Yaskawa INFORM job: DEMO_ROOF_SIDE_0625_3PAINT_5.JBI

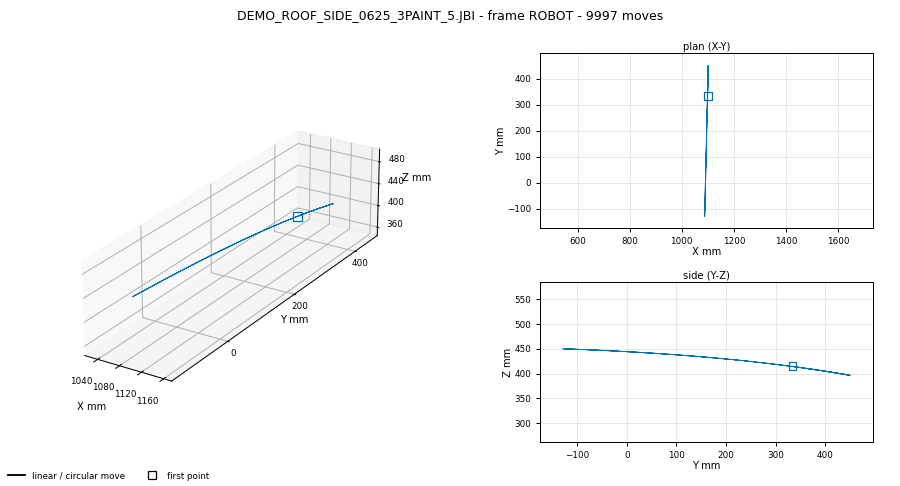
[picture p0: tool path of DEMO_ROOF_SIDE_0625_3PAINT_5.JBI in frame ROBOT, 9997 of 9997 moves have a stored position in this frame; points joined in program order, loops and branches not executed]
/JOB
//NAME DEMO_ROOF_SIDE_0625_3PAINT5
//POS
///NPOS 9997,0,0,0,0,0
///TOOL 0
///USER 0
///POSTYPE ROBOT
///RECTAN
///RCONF 1,0,0,0,0,0,0,0,0,0,0,0,0,0,0,0,0,0,0,0,0,0,0,0
C00000=1099.831,334.377,414.802,179.080,18.325,152.124
C00001=1099.836,334.624,414.769,179.083,18.328,152.124
C00002=1099.842,334.872,414.736,179.086,18.331,152.124
C00003=1099.847,335.120,414.703,179.089,18.334,152.124
C00004=1099.853,335.368,414.670,179.092,18.337,152.124
C00005=1099.859,335.615,414.637,179.095,18.340,152.124
C00006=1099.865,335.863,414.604,179.099,18.343,152.124
C00007=1099.870,336.112,414.571,179.102,18.346,152.125
C00008=1099.876,336.359,414.539,179.105,18.349,152.125
C00009=1099.881,336.607,414.505,179.109,18.352,152.125
C00010=1099.887,336.855,414.472,179.112,18.355,152.125
C00011=1099.893,337.102,414.439,179.115,18.358,152.125
C00012=1099.899,337.350,414.406,179.118,18.361,152.125
C00013=1099.904,337.598,414.372,179.121,18.364,152.125
C00014=1099.910,337.845,414.338,179.124,18.367,152.125
C00015=1099.916,338.093,414.306,179.127,18.370,152.125
C00016=1099.922,338.341,414.272,179.131,18.373,152.126
C00017=1099.928,338.589,414.239,179.134,18.376,152.126
C00018=1099.933,338.837,414.206,179.137,18.379,152.126
C00019=1099.939,339.084,414.172,179.140,18.382,152.126
C00020=1099.945,339.332,414.140,179.143,18.385,152.126
C00021=1099.951,339.580,414.106,179.146,18.388,152.126
C00022=1099.956,339.827,414.072,179.150,18.392,152.127
C00023=1099.961,340.074,414.039,179.153,18.395,152.127
C00024=1099.967,340.322,414.006,179.156,18.397,152.127
C00025=1099.972,340.570,413.973,179.159,18.401,152.127
C00026=1099.978,340.818,413.939,179.162,18.404,152.127
C00027=1099.984,341.065,413.905,179.165,18.407,152.127
C00028=1099.989,341.313,413.872,179.168,18.411,152.128
C00029=1099.996,341.561,413.839,179.171,18.413,152.128
C00030=1100.001,341.809,413.806,179.175,18.417,152.128
C00031=1100.007,342.056,413.772,179.178,18.420,152.128
C00032=1100.013,342.304,413.738,179.181,18.423,152.128
C00033=1100.018,342.552,413.705,179.184,18.427,152.128
C00034=1100.027,342.925,413.654,179.189,18.431,152.129
C00035=1100.036,343.298,413.603,179.194,18.436,152.129
C00036=1100.044,343.671,413.552,179.199,18.441,152.129
C00037=1100.053,344.044,413.502,179.203,18.446,152.129
C00038=1100.059,344.291,413.469,179.207,18.449,152.130
C00039=1100.065,344.539,413.435,179.209,18.452,152.130
C00040=1100.070,344.787,413.401,179.212,18.455,152.130
C00041=1100.076,345.034,413.367,179.216,18.459,152.130
C00042=1100.082,345.283,413.333,179.219,18.462,152.130
C00043=1100.087,345.530,413.299,179.222,18.466,152.131
C00044=1100.093,345.778,413.266,179.225,18.469,152.131
C00045=1100.099,346.025,413.231,179.228,18.472,152.131
C00046=1100.104,346.273,413.198,179.231,18.475,152.131
C00047=1100.110,346.520,413.164,179.234,18.479,152.132
C00048=1100.116,346.768,413.130,179.238,18.482,152.132
C00049=1100.121,347.016,413.097,179.240,18.486,152.132
C00050=1100.127,347.263,413.062,179.244,18.489,152.132
C00051=1100.132,347.511,413.029,179.247,18.492,152.132
C00052=1100.138,347.758,412.995,179.249,18.495,152.133
C00053=1100.144,348.006,412.960,179.253,18.499,152.133
C00054=1100.150,348.254,412.926,179.256,18.502,152.133
C00055=1100.156,348.502,412.893,179.259,18.506,152.133
C00056=1100.161,348.749,412.858,179.262,18.509,152.134
C00057=1100.167,348.997,412.824,179.265,18.513,152.134
C00058=1100.172,349.244,412.791,179.268,18.516,152.134
C00059=1100.178,349.492,412.757,179.272,18.520,152.134
C00060=1100.184,349.740,412.722,179.274,18.523,152.135
C00061=1100.190,349.987,412.688,179.278,18.527,152.135
C00062=1100.196,350.235,412.654,179.281,18.530,152.135
C00063=1100.201,350.482,412.619,179.284,18.534,152.135
C00064=1100.206,350.730,412.586,179.287,18.537,152.136
C00065=1100.212,350.977,412.552,179.290,18.541,152.136
C00066=1100.219,351.225,412.517,179.293,18.544,152.136
C00067=1100.224,351.473,412.483,179.296,18.548,152.136
C00068=1100.230,351.720,412.448,179.299,18.551,152.137
C00069=1100.236,351.967,412.414,179.302,18.555,152.137
C00070=1100.241,352.215,412.380,179.305,18.558,152.137
C00071=1100.247,352.463,412.345,179.309,18.562,152.138
C00072=1100.253,352.710,412.311,179.311,18.565,152.138
C00073=1100.258,352.958,412.277,179.315,18.569,152.138
C00074=1100.264,353.205,412.243,179.318,18.572,152.139
C00075=1100.270,353.454,412.208,179.321,18.577,152.139
C00076=1100.276,353.701,412.174,179.323,18.580,152.139
C00077=1100.281,353.948,412.139,179.327,18.584,152.139
C00078=1100.287,354.196,412.105,179.329,18.587,152.140
C00079=1100.293,354.444,412.070,179.333,18.591,152.140
C00080=1100.298,354.691,412.036,179.336,18.594,152.140
C00081=1100.304,354.939,412.002,179.339,18.598,152.141
C00082=1100.309,355.186,411.967,179.342,18.602,152.141
C00083=1100.316,355.434,411.932,179.345,18.606,152.141
C00084=1100.321,355.681,411.897,179.348,18.609,152.142
C00085=1100.327,355.928,411.863,179.351,18.613,152.142
C00086=1100.335,356.304,411.810,179.356,18.619,152.143
C00087=1100.344,356.679,411.758,179.360,18.625,152.143
C00088=1100.353,357.055,411.706,179.365,18.630,152.144
C00089=1100.361,357.430,411.653,179.369,18.636,152.144
C00090=1100.367,357.678,411.618,179.372,18.639,152.144
C00091=1100.373,357.925,411.583,179.375,18.644,152.145
C00092=1100.378,358.172,411.548,179.378,18.647,152.145
C00093=1100.384,358.420,411.514,179.381,18.651,152.146
C00094=1100.390,358.667,411.479,179.385,18.655,152.146
C00095=1100.396,358.914,411.445,179.387,18.659,152.146
C00096=1100.402,359.162,411.409,179.391,18.663,152.147
C00097=1100.407,359.410,411.374,179.393,18.666,152.147
C00098=1100.413,359.658,411.340,179.396,18.670,152.148
C00099=1100.419,359.905,411.304,179.399,18.675,152.148
C00100=1100.425,360.152,411.270,179.402,18.678,152.148
C00101=1100.431,360.400,411.235,179.405,18.682,152.149
C00102=1100.436,360.647,411.200,179.409,18.686,152.149
C00103=1100.441,360.894,411.165,179.411,18.690,152.149
C00104=1100.448,361.142,411.130,179.414,18.694,152.150
C00105=1100.453,361.389,411.095,179.417,18.698,152.150
C00106=1100.459,361.637,411.060,179.420,18.702,152.151
C00107=1100.464,361.884,411.024,179.423,18.706,152.151
C00108=1100.470,362.131,410.990,179.426,18.710,152.152
C00109=1100.476,362.379,410.955,179.429,18.714,152.152
C00110=1100.482,362.626,410.919,179.432,18.718,152.152
C00111=1100.488,362.874,410.884,179.435,18.722,152.153
C00112=1100.493,363.121,410.850,179.438,18.726,152.153
C00113=1100.499,363.369,410.814,179.441,18.730,152.154
C00114=1100.505,363.616,410.778,179.444,18.734,152.154
C00115=1100.510,363.863,410.744,179.447,18.738,152.154
C00116=1100.516,364.111,410.708,179.450,18.743,152.155
C00117=1100.521,364.358,410.673,179.452,18.746,152.155
C00118=1100.528,364.606,410.638,179.456,18.751,152.156
C00119=1100.533,364.853,410.603,179.459,18.755,152.156
C00120=1100.539,365.101,410.567,179.461,18.758,152.157
C00121=1100.545,365.348,410.532,179.464,18.763,152.157
C00122=1100.551,365.595,410.496,179.468,18.767,152.158
C00123=1100.556,365.842,410.461,179.470,18.771,152.158
C00124=1100.562,366.091,410.426,179.473,18.775,152.159
C00125=1100.567,366.338,410.390,179.476,18.780,152.159
C00126=1100.573,366.585,410.355,179.479,18.784,152.160
C00127=1100.579,366.832,410.319,179.482,18.788,152.160
C00128=1100.585,367.080,410.284,179.485,18.792,152.161
C00129=1100.590,367.327,410.248,179.488,18.797,152.161
C00130=1100.596,367.575,410.212,179.490,18.801,152.162
C00131=1100.602,367.822,410.177,179.494,18.805,152.162
C00132=1100.608,368.069,410.141,179.497,18.809,152.163
C00133=1100.613,368.316,410.106,179.500,18.814,152.163
C00134=1100.619,368.564,410.070,179.502,18.818,152.164
C00135=1100.625,368.811,410.035,179.505,18.822,152.164
C00136=1100.631,369.059,409.999,179.508,18.827,152.165
C00137=1100.636,369.306,409.964,179.511,18.832,152.165
C00138=1100.645,369.696,409.908,179.516,18.838,152.166
C00139=1100.654,370.086,409.851,179.520,18.845,152.167
C00140=1100.664,370.476,409.794,179.524,18.852,152.168
C00141=1100.672,370.867,409.738,179.529,18.859,152.169
C00142=1100.678,371.114,409.702,179.532,18.863,152.169
C00143=1100.684,371.362,409.666,179.535,18.867,152.170
C00144=1100.689,371.609,409.631,179.538,18.872,152.170
C00145=1100.695,371.856,409.595,179.541,18.877,152.171
C00146=1100.701,372.103,409.559,179.544,18.881,152.171
C00147=1100.707,372.350,409.524,179.546,18.885,152.172
C00148=1100.712,372.598,409.487,179.549,18.890,152.173
C00149=1100.718,372.845,409.451,179.552,18.895,152.173
C00150=1100.724,373.092,409.415,179.555,18.899,152.174
C00151=1100.730,373.340,409.380,179.558,18.904,152.174
C00152=1100.736,373.586,409.344,179.560,18.908,152.175
C00153=1100.741,373.834,409.307,179.563,18.913,152.176
C00154=1100.747,374.082,409.271,179.566,18.917,152.176
C00155=1100.753,374.329,409.236,179.569,18.922,152.177
C00156=1100.759,374.576,409.200,179.572,18.927,152.177
C00157=1100.764,374.824,409.163,179.575,18.932,152.178
C00158=1100.770,375.071,409.127,179.577,18.936,152.179
C00159=1100.776,375.318,409.091,179.580,18.941,152.179
C00160=1100.781,375.566,409.055,179.583,18.945,152.180
C00161=1100.787,375.812,409.019,179.586,18.950,152.181
C00162=1100.792,376.060,408.982,179.589,18.955,152.181
C00163=1100.799,376.307,408.946,179.592,18.960,152.182
C00164=1100.804,376.554,408.910,179.595,18.965,152.182
C00165=1100.810,376.801,408.873,179.597,18.970,152.183
C00166=1100.816,377.049,408.838,179.600,18.974,152.184
C00167=1100.821,377.296,408.801,179.602,18.979,152.184
C00168=1100.827,377.543,408.765,179.605,18.984,152.185
C00169=1100.832,377.791,408.728,179.608,18.988,152.186
C00170=1100.838,378.037,408.692,179.611,18.993,152.186
C00171=1100.845,378.284,408.656,179.614,18.998,152.187
C00172=1100.850,378.532,408.619,179.617,19.003,152.188
C00173=1100.856,378.779,408.583,179.620,19.008,152.188
C00174=1100.861,379.026,408.546,179.622,19.013,152.189
C00175=1100.867,379.273,408.510,179.625,19.018,152.190
C00176=1100.873,379.521,408.473,179.627,19.022,152.191
C00177=1100.879,379.768,408.437,179.630,19.027,152.191
C00178=1100.884,380.015,408.400,179.633,19.032,152.192
C00179=1100.890,380.262,408.364,179.636,19.037,152.193
C00180=1100.896,380.510,408.328,179.638,19.042,152.193
C00181=1100.902,380.757,408.291,179.641,19.047,152.194
C00182=1100.908,381.004,408.254,179.644,19.052,152.195
C00183=1100.913,381.250,408.218,179.647,19.057,152.196
C00184=1100.919,381.498,408.181,179.649,19.062,152.196
C00185=1100.925,381.745,408.144,179.652,19.068,152.197
C00186=1100.931,381.992,408.107,179.655,19.073,152.198
C00187=1100.937,382.239,408.070,179.658,19.078,152.199
C00188=1100.943,382.487,408.034,179.661,19.083,152.199
C00189=1100.948,382.733,407.997,179.663,19.088,152.200
C00190=1100.958,383.151,407.936,179.668,19.096,152.201
C00191=1100.967,383.568,407.873,179.673,19.105,152.203
C00192=1100.978,383.985,407.811,179.677,19.114,152.204
C00193=1100.987,384.403,407.749,179.682,19.123,152.205
C00194=1100.992,384.650,407.712,179.684,19.128,152.206
C00195=1100.998,384.897,407.675,179.687,19.133,152.207
C00196=1101.004,385.144,407.637,179.689,19.139,152.208
C00197=1101.010,385.391,407.601,179.692,19.144,152.209
C00198=1101.016,385.638,407.564,179.695,19.149,152.209
C00199=1101.021,385.885,407.527,179.697,19.155,152.210
C00200=1101.027,386.133,407.490,179.700,19.160,152.211
C00201=1101.032,386.380,407.453,179.703,19.165,152.212
C00202=1101.038,386.626,407.416,179.705,19.170,152.213
C00203=1101.044,386.873,407.379,179.708,19.176,152.214
C00204=1101.050,387.121,407.342,179.710,19.181,152.214
C00205=1101.055,387.367,407.304,179.713,19.187,152.215
C00206=1101.061,387.615,407.267,179.716,19.192,152.216
C00207=1101.067,387.862,407.230,179.719,19.198,152.217
C00208=1101.073,388.109,407.193,179.721,19.203,152.218
C00209=1101.079,388.356,407.156,179.724,19.209,152.219
C00210=1101.084,388.603,407.119,179.727,19.214,152.220
C00211=1101.090,388.850,407.081,179.729,19.220,152.220
C00212=1101.096,389.097,407.044,179.732,19.225,152.221
C00213=1101.102,389.345,407.007,179.734,19.230,152.222
C00214=1101.108,389.592,406.969,179.737,19.236,152.223
C00215=1101.113,389.839,406.932,179.739,19.242,152.224
C00216=1101.119,390.086,406.895,179.743,19.248,152.225
C00217=1101.125,390.333,406.857,179.745,19.253,152.226
C00218=1101.131,390.579,406.820,179.748,19.258,152.227
C00219=1101.137,390.827,406.783,179.750,19.264,152.228
C00220=1101.143,391.074,406.746,179.753,19.270,152.229
C00221=1101.149,391.320,406.708,179.755,19.276,152.230
C00222=1101.154,391.568,406.671,179.758,19.281,152.230
C00223=1101.160,391.814,406.633,179.761,19.287,152.231
C00224=1101.166,392.062,406.596,179.763,19.293,152.232
C00225=1101.172,392.308,406.558,179.766,19.299,152.233
C00226=1101.178,392.555,406.520,179.768,19.304,152.234
C00227=1101.183,392.803,406.483,179.770,19.310,152.235
C00228=1101.189,393.049,406.446,179.773,19.316,152.236
C00229=1101.194,393.296,406.407,179.776,19.322,152.237
C00230=1101.200,393.544,406.370,179.779,19.327,152.238
C00231=1101.206,393.790,406.332,179.781,19.333,152.239
C00232=1101.212,394.038,406.294,179.783,19.339,152.240
C00233=1101.218,394.285,406.257,179.786,19.345,152.241
C00234=1101.224,394.532,406.220,179.789,19.351,152.242
C00235=1101.229,394.779,406.181,179.791,19.357,152.243
C00236=1101.235,395.026,406.143,179.793,19.363,152.244
C00237=1101.241,395.273,406.106,179.796,19.369,152.245
C00238=1101.246,395.520,406.069,179.799,19.375,152.246
C00239=1101.253,395.767,406.031,179.801,19.381,152.247
C00240=1101.258,396.014,405.992,179.803,19.387,152.248
C00241=1101.264,396.261,405.954,179.806,19.393,152.249
C00242=1101.269,396.476,405.922,179.808,19.398,152.250
C00243=1101.274,396.690,405.889,179.810,19.403,152.251
C00244=1101.279,396.906,405.856,179.812,19.409,152.252
C00245=1101.284,397.121,405.823,179.815,19.415,152.253
C00246=1101.289,397.335,405.789,179.817,19.419,152.254
C00247=1101.294,397.550,405.756,179.819,19.425,152.255
C00248=1101.299,397.765,405.723,179.821,19.430,152.256
C00249=1101.304,397.980,405.690,179.823,19.436,152.257
C00250=1101.309,398.227,405.652,179.825,19.442,152.258
C00251=1101.315,398.473,405.614,179.828,19.448,152.259
C00252=1101.322,398.721,405.576,179.830,19.455,152.260
C00253=1101.327,398.968,405.538,179.833,19.460,152.261
C00254=1101.333,399.215,405.500,179.836,19.467,152.262
C00255=1101.339,399.461,405.462,179.838,19.473,152.264
C00256=1101.344,399.709,405.424,179.840,19.480,152.265
C00257=1101.351,399.955,405.385,179.843,19.486,152.266
C00258=1101.356,400.202,405.347,179.845,19.492,152.267
C00259=1101.362,400.449,405.309,179.847,19.498,152.268
C00260=1101.367,400.697,405.270,179.850,19.506,152.269
C00261=1101.373,400.944,405.232,179.852,19.512,152.271
C00262=1101.378,401.191,405.194,179.854,19.518,152.272
C00263=1101.385,401.437,405.155,179.857,19.525,152.273
C00264=1101.390,401.685,405.117,179.859,19.531,152.274
C00265=1101.396,401.931,405.079,179.862,19.538,152.275
C00266=1101.402,402.179,405.040,179.864,19.544,152.276
C00267=1101.408,402.425,405.002,179.866,19.551,152.278
C00268=1101.414,402.672,404.964,179.869,19.557,152.279
C00269=1101.419,402.920,404.925,179.871,19.564,152.280
C00270=1101.426,403.166,404.886,179.874,19.571,152.281
C00271=1101.431,403.413,404.848,179.876,19.577,152.283
C00272=1101.437,403.660,404.809,179.879,19.584,152.284
C00273=1101.443,403.907,404.771,179.881,19.591,152.285
C00274=1101.448,404.154,404.733,179.884,19.598,152.286
C00275=1101.455,404.401,404.694,179.886,19.604,152.287
C00276=1101.460,404.648,404.655,179.888,19.611,152.289
C00277=1101.466,404.895,404.616,179.891,19.618,152.290
C00278=1101.472,405.142,404.578,179.893,19.625,152.291
C00279=1101.477,405.388,404.539,179.895,19.631,152.292
C00280=1101.483,405.636,404.500,179.898,19.638,152.294
C00281=1101.489,405.882,404.462,179.900,19.645,152.295
C00282=1101.495,406.130,404.423,179.903,19.652,152.296
C00283=1101.500,406.376,404.384,179.905,19.659,152.298
C00284=1101.506,406.623,404.345,179.907,19.666,152.299
C00285=1101.512,406.870,404.307,179.909,19.673,152.300
C00286=1101.518,407.117,404.268,179.912,19.680,152.302
C00287=1101.524,407.364,404.229,179.914,19.687,152.303
C00288=1101.529,407.611,404.190,179.916,19.694,152.304
C00289=1101.535,407.858,404.151,179.919,19.702,152.306
C00290=1101.541,408.104,404.112,179.921,19.708,152.307
C00291=1101.547,408.352,404.074,179.923,19.716,152.309
C00292=1101.553,408.598,404.034,179.925,19.722,152.310
C00293=1101.558,408.845,403.995,179.928,19.730,152.311
C00294=1101.564,409.092,403.956,179.930,19.738,152.313
C00295=1101.569,409.339,403.918,179.932,19.744,152.314
C00296=1101.575,409.586,403.878,179.935,19.752,152.315
C00297=1101.581,409.832,403.839,179.937,19.759,152.317
C00298=1101.587,410.048,403.805,179.939,19.765,152.318
C00299=1101.591,410.263,403.771,179.941,19.772,152.319
C00300=1101.596,410.478,403.737,179.942,19.778,152.321
C00301=1101.601,410.693,403.703,179.945,19.784,152.322
C00302=1101.606,410.906,403.668,179.947,19.791,152.323
C00303=1101.612,411.122,403.634,179.949,19.797,152.324
C00304=1101.616,411.336,403.600,179.950,19.804,152.326
C00305=1101.622,411.552,403.566,179.953,19.810,152.327
C00306=1101.627,411.798,403.527,179.955,19.818,152.328
C00307=1101.633,412.045,403.488,179.957,19.826,152.330
C00308=1101.639,412.292,403.449,179.959,19.833,152.331
C00309=1101.645,412.539,403.409,179.962,19.840,152.333
C00310=1101.651,412.786,403.370,179.964,19.848,152.334
C00311=1101.656,413.032,403.331,179.967,19.856,152.336
C00312=1101.662,413.280,403.291,179.969,19.864,152.337
C00313=1101.667,413.526,403.252,179.971,19.871,152.339
C00314=1101.673,413.773,403.212,179.973,19.879,152.340
C00315=1101.680,414.020,403.172,179.975,19.886,152.342
C00316=1101.685,414.266,403.133,179.978,19.894,152.343
C00317=1101.691,414.513,403.094,179.980,19.902,152.345
C00318=1101.697,414.761,403.054,179.982,19.909,152.346
C00319=1101.703,415.006,403.014,179.984,19.917,152.348
C00320=1101.709,415.253,402.975,179.986,19.925,152.350
C00321=1101.715,415.501,402.936,179.989,19.933,152.351
C00322=1101.721,415.747,402.896,179.991,19.941,152.353
C00323=1101.726,415.994,402.856,179.993,19.949,152.354
C00324=1101.732,416.241,402.816,179.995,19.956,152.356
C00325=1101.738,416.487,402.777,179.997,19.964,152.358
C00326=1101.744,416.734,402.737,180.000,19.972,152.359
C00327=1101.750,416.981,402.698,-179.998,19.981,152.361
C00328=1101.755,417.227,402.657,-179.996,19.989,152.362
C00329=1101.761,417.474,402.618,-179.994,19.997,152.364
C00330=1101.767,417.721,402.578,-179.991,20.005,152.366
C00331=1101.772,417.968,402.538,-179.989,20.013,152.367
C00332=1101.779,418.215,402.499,-179.987,20.022,152.369
C00333=1101.785,418.461,402.458,-179.985,20.030,152.371
C00334=1101.790,418.708,402.419,-179.983,20.038,152.372
C00335=1101.796,418.955,402.379,-179.981,20.046,152.374
C00336=1101.802,419.201,402.338,-179.978,20.055,152.376
C00337=1101.808,419.448,402.298,-179.976,20.063,152.378
C00338=1101.813,419.694,402.259,-179.974,20.071,152.379
C00339=1101.819,419.942,402.219,-179.972,20.080,152.381
C00340=1101.825,420.188,402.179,-179.970,20.088,152.383
C00341=1101.832,420.435,402.138,-179.968,20.096,152.385
C00342=1101.836,420.682,402.099,-179.966,20.105,152.386
C00343=1101.843,420.928,402.059,-179.964,20.113,152.388
C00344=1101.848,421.175,402.018,-179.962,20.122,152.390
C00345=1101.855,421.421,401.978,-179.959,20.130,152.392
C00346=1101.860,421.669,401.938,-179.958,20.139,152.393
C00347=1101.866,421.915,401.898,-179.955,20.147,152.395
C00348=1101.872,422.161,401.858,-179.954,20.156,152.397
C00349=1101.878,422.408,401.817,-179.952,20.165,152.399
C00350=1101.884,422.654,401.777,-179.949,20.173,152.401
C00351=1101.890,422.902,401.737,-179.947,20.182,152.402
C00352=1101.896,423.148,401.697,-179.946,20.191,152.404
C00353=1101.901,423.395,401.656,-179.943,20.200,152.406
C00354=1101.906,423.616,401.620,-179.941,20.208,152.408
C00355=1101.911,423.838,401.583,-179.939,20.216,152.410
C00356=1101.917,424.059,401.547,-179.938,20.223,152.411
C00357=1101.922,424.281,401.511,-179.936,20.232,152.413
C00358=1101.927,424.503,401.474,-179.934,20.239,152.415
C00359=1101.932,424.724,401.437,-179.932,20.248,152.416
C00360=1101.938,424.946,401.402,-179.931,20.256,152.418
C00361=1101.943,425.167,401.365,-179.928,20.264,152.420
C00362=1101.949,425.414,401.324,-179.927,20.273,152.422
C00363=1101.955,425.661,401.284,-179.925,20.282,152.424
C00364=1101.960,425.907,401.244,-179.922,20.291,152.426
C00365=1101.966,426.154,401.203,-179.920,20.301,152.428
C00366=1101.972,426.401,401.162,-179.919,20.310,152.430
C00367=1101.978,426.647,401.122,-179.917,20.319,152.432
C00368=1101.984,426.893,401.080,-179.914,20.328,152.434
C00369=1101.989,427.140,401.040,-179.912,20.337,152.436
C00370=1101.996,427.387,401.000,-179.911,20.346,152.438
C00371=1102.001,427.633,400.959,-179.909,20.356,152.440
C00372=1102.007,427.880,400.917,-179.907,20.366,152.442
C00373=1102.013,428.126,400.877,-179.905,20.375,152.444
C00374=1102.019,428.373,400.836,-179.903,20.384,152.446
C00375=1102.025,428.619,400.795,-179.901,20.394,152.448
C00376=1102.031,428.866,400.754,-179.899,20.403,152.450
C00377=1102.037,429.113,400.714,-179.897,20.413,152.452
C00378=1102.043,429.359,400.672,-179.896,20.422,152.454
C00379=1102.048,429.605,400.632,-179.893,20.432,152.456
C00380=1102.054,429.851,400.591,-179.892,20.442,152.458
C00381=1102.060,430.098,400.550,-179.890,20.451,152.460
C00382=1102.066,430.344,400.509,-179.888,20.461,152.463
C00383=1102.072,430.591,400.468,-179.886,20.471,152.465
C00384=1102.078,430.837,400.426,-179.884,20.481,152.467
C00385=1102.083,431.084,400.386,-179.882,20.490,152.469
C00386=1102.089,431.330,400.344,-179.881,20.500,152.471
C00387=1102.095,431.577,400.303,-179.878,20.510,152.473
C00388=1102.101,431.823,400.262,-179.877,20.520,152.475
C00389=1102.107,432.069,400.221,-179.875,20.530,152.478
C00390=1102.112,432.316,400.180,-179.873,20.540,152.480
C00391=1102.118,432.562,400.138,-179.871,20.550,152.482
C00392=1102.125,432.809,400.097,-179.869,20.560,152.484
C00393=1102.130,433.056,400.056,-179.868,20.570,152.487
C00394=1102.136,433.302,400.014,-179.866,20.581,152.489
C00395=1102.142,433.549,399.973,-179.864,20.591,152.491
C00396=1102.148,433.795,399.931,-179.862,20.601,152.494
C00397=1102.154,434.041,399.890,-179.861,20.611,152.496
C00398=1102.160,434.288,399.849,-179.859,20.621,152.498
C00399=1102.165,434.534,399.807,-179.857,20.632,152.500
C00400=1102.171,434.781,399.766,-179.855,20.642,152.503
C00401=1102.177,435.027,399.724,-179.853,20.653,152.505
C00402=1102.183,435.273,399.683,-179.852,20.663,152.508
C00403=1102.189,435.519,399.641,-179.850,20.674,152.510
C00404=1102.194,435.766,399.599,-179.848,20.684,152.512
C00405=1102.200,436.012,399.558,-179.846,20.695,152.515
C00406=1102.206,436.258,399.516,-179.845,20.705,152.517
C00407=1102.213,436.505,399.475,-179.843,20.716,152.520
C00408=1102.218,436.751,399.433,-179.842,20.727,152.522
C00409=1102.224,436.998,399.391,-179.840,20.738,152.524
C00410=1102.233,437.381,399.326,-179.838,20.755,152.528
C00411=1102.242,437.764,399.261,-179.835,20.772,152.532
C00412=1102.251,438.148,399.196,-179.832,20.788,152.536
C00413=1102.260,438.531,399.131,-179.830,20.805,152.540
C00414=1102.266,438.778,399.089,-179.828,20.817,152.542
C00415=1102.273,439.023,399.047,-179.826,20.827,152.545
C00416=1102.278,439.270,399.005,-179.825,20.839,152.548
C00417=1102.284,439.517,398.963,-179.823,20.850,152.550
C00418=1102.291,439.762,398.921,-179.822,20.861,152.553
C00419=1102.297,440.008,398.880,-179.821,20.872,152.555
C00420=1102.302,440.255,398.838,-179.819,20.883,152.558
C00421=1102.309,440.501,398.795,-179.817,20.895,152.560
C00422=1102.314,440.748,398.753,-179.815,20.906,152.563
C00423=1102.320,440.993,398.711,-179.814,20.917,152.566
C00424=1102.325,441.240,398.669,-179.813,20.929,152.568
C00425=1102.332,441.487,398.627,-179.811,20.940,152.571
C00426=1102.337,441.733,398.584,-179.809,20.952,152.574
C00427=1102.343,441.979,398.543,-179.808,20.963,152.576
C00428=1102.349,442.225,398.500,-179.807,20.975,152.579
C00429=1102.355,442.472,398.458,-179.805,20.987,152.582
C00430=1102.361,442.717,398.415,-179.803,20.999,152.584
C00431=1102.367,442.963,398.373,-179.802,21.011,152.587
C00432=1102.372,443.210,398.331,-179.800,21.023,152.590
C00433=1102.379,443.456,398.289,-179.799,21.034,152.593
C00434=1102.385,443.702,398.246,-179.798,21.046,152.596
C00435=1102.390,443.948,398.204,-179.796,21.058,152.598
C00436=1102.397,444.195,398.161,-179.796,21.070,152.601
C00437=1102.402,444.440,398.119,-179.795,21.081,152.604
C00438=1102.408,444.686,398.076,-179.794,21.094,152.607
C00439=1102.414,444.933,398.034,-179.793,21.105,152.610
C00440=1102.420,445.179,397.991,-179.793,21.117,152.613
C00441=1102.426,445.426,397.948,-179.793,21.128,152.616
C00442=1102.432,445.671,397.906,-179.792,21.140,152.619
C00443=1102.437,445.918,397.864,-179.793,21.152,152.622
C00444=1102.444,446.164,397.821,-179.792,21.164,152.625
C00445=1102.449,446.410,397.778,-179.793,21.175,152.628
C00446=1102.456,446.657,397.735,-179.793,21.187,152.631
C00447=1102.461,446.902,397.693,-179.794,21.199,152.634
C00448=1102.467,447.148,397.650,-179.794,21.210,152.637
C00449=1102.473,447.395,397.607,-179.795,21.222,152.640
C00450=1102.479,447.641,397.564,-179.795,21.234,152.643
C00451=1102.485,447.887,397.521,-179.796,21.245,152.646
C00452=1102.491,448.134,397.479,-179.797,21.257,152.649
C00453=1102.497,448.380,397.436,-179.798,21.268,152.652
C00454=1102.502,448.626,397.393,-179.800,21.280,152.656
C00455=1102.508,448.873,397.350,-179.801,21.291,152.659
C00456=1102.514,449.119,397.308,-179.802,21.304,152.662
C00457=1102.520,449.365,397.264,-179.804,21.315,152.665
C00458=1102.526,449.611,397.222,-179.806,21.326,152.668
C00459=1102.532,449.856,397.179,-179.807,21.338,152.671
C00460=1102.538,450.103,397.136,-179.809,21.349,152.675
C00461=1102.544,450.349,397.092,-179.810,21.361,152.678
C00462=1102.144,450.341,396.956,-179.881,21.585,152.746
C00463=1102.137,450.095,396.998,-179.879,21.574,152.743
C00464=1102.131,449.849,397.041,-179.878,21.562,152.740
C00465=1102.126,449.603,397.084,-179.876,21.551,152.737
C00466=1102.120,449.356,397.127,-179.874,21.540,152.733
C00467=1102.114,449.110,397.170,-179.872,21.528,152.730
C00468=1102.107,448.864,397.212,-179.871,21.516,152.727
C00469=1102.101,448.619,397.256,-179.871,21.504,152.724
C00470=1102.095,448.372,397.299,-179.869,21.493,152.721
C00471=1102.090,448.126,397.341,-179.868,21.481,152.718
C00472=1102.084,447.880,397.385,-179.868,21.469,152.715
C00473=1102.078,447.634,397.427,-179.866,21.458,152.711
C00474=1102.072,447.387,397.471,-179.866,21.446,152.708
C00475=1102.066,447.141,397.513,-179.865,21.434,152.705
C00476=1102.060,446.895,397.556,-179.865,21.422,152.702
C00477=1102.054,446.648,397.598,-179.865,21.411,152.699
C00478=1102.048,446.402,397.641,-179.864,21.399,152.696
C00479=1102.043,446.156,397.684,-179.864,21.387,152.693
C00480=1102.037,445.910,397.727,-179.863,21.375,152.690
C00481=1102.030,445.664,397.769,-179.864,21.363,152.687
C00482=1102.025,445.418,397.812,-179.865,21.351,152.684
C00483=1102.019,445.171,397.855,-179.864,21.340,152.681
C00484=1102.013,444.926,397.897,-179.865,21.328,152.678
C00485=1102.006,444.679,397.940,-179.866,21.316,152.675
C00486=1102.001,444.433,397.982,-179.866,21.304,152.672
C00487=1101.995,444.187,398.025,-179.868,21.292,152.669
C00488=1101.989,443.940,398.068,-179.868,21.280,152.667
C00489=1101.983,443.694,398.110,-179.870,21.268,152.664
C00490=1101.977,443.448,398.152,-179.871,21.256,152.661
C00491=1101.971,443.202,398.195,-179.872,21.244,152.658
C00492=1101.966,442.956,398.238,-179.874,21.232,152.655
C00493=1101.959,442.710,398.280,-179.876,21.221,152.653
C00494=1101.954,442.463,398.322,-179.877,21.209,152.650
C00495=1101.947,442.217,398.365,-179.879,21.197,152.647
C00496=1101.942,441.971,398.407,-179.880,21.186,152.644
C00497=1101.935,441.725,398.449,-179.882,21.174,152.642
C00498=1101.930,441.479,398.492,-179.883,21.162,152.639
C00499=1101.924,441.232,398.533,-179.885,21.150,152.636
C00500=1101.918,440.987,398.576,-179.887,21.139,152.634
C00501=1101.912,440.740,398.618,-179.888,21.127,152.631
C00502=1101.906,440.494,398.661,-179.890,21.116,152.628
C00503=1101.900,440.248,398.702,-179.892,21.104,152.626
C00504=1101.895,440.000,398.745,-179.894,21.093,152.623
C00505=1101.888,439.755,398.787,-179.894,21.082,152.620
C00506=1101.882,439.509,398.828,-179.896,21.071,152.618
C00507=1101.877,439.263,398.871,-179.898,21.059,152.615
C00508=1101.870,439.016,398.913,-179.899,21.048,152.613
C00509=1101.864,438.770,398.954,-179.901,21.037,152.610
C00510=1101.859,438.524,398.997,-179.903,21.026,152.608
C00511=1101.850,438.147,399.061,-179.906,21.009,152.604
C00512=1101.841,437.770,399.125,-179.908,20.992,152.600
C00513=1101.832,437.393,399.189,-179.911,20.975,152.596
C00514=1101.823,437.017,399.252,-179.913,20.959,152.592
C00515=1101.816,436.770,399.294,-179.915,20.948,152.590
C00516=1101.811,436.523,399.336,-179.917,20.938,152.588
C00517=1101.805,436.277,399.378,-179.918,20.926,152.585
C00518=1101.799,436.031,399.420,-179.921,20.916,152.583
C00519=1101.793,435.785,399.461,-179.922,20.905,152.580
C00520=1101.787,435.539,399.503,-179.924,20.894,152.578
C00521=1101.782,435.292,399.545,-179.925,20.884,152.575
C00522=1101.776,435.046,399.586,-179.927,20.873,152.573
C00523=1101.769,434.799,399.628,-179.929,20.863,152.571
C00524=1101.764,434.552,399.669,-179.931,20.852,152.568
C00525=1101.758,434.306,399.711,-179.933,20.842,152.566
C00526=1101.752,434.060,399.752,-179.934,20.831,152.564
C00527=1101.746,433.814,399.794,-179.937,20.821,152.561
C00528=1101.740,433.567,399.835,-179.938,20.810,152.559
C00529=1101.734,433.321,399.877,-179.940,20.800,152.557
C00530=1101.728,433.075,399.918,-179.942,20.790,152.554
C00531=1101.723,432.828,399.959,-179.943,20.780,152.552
C00532=1101.717,432.582,400.000,-179.946,20.770,152.550
C00533=1101.711,432.336,400.042,-179.947,20.760,152.548
C00534=1101.705,432.090,400.083,-179.949,20.749,152.545
C00535=1101.699,431.843,400.124,-179.951,20.740,152.543
C00536=1101.693,431.596,400.166,-179.953,20.729,152.541
C00537=1101.687,431.350,400.207,-179.955,20.719,152.539
C00538=1101.681,431.103,400.248,-179.956,20.710,152.537
C00539=1101.675,430.857,400.289,-179.959,20.699,152.534
C00540=1101.670,430.610,400.330,-179.960,20.690,152.532
C00541=1101.664,430.364,400.372,-179.963,20.680,152.530
C00542=1101.658,430.117,400.413,-179.964,20.670,152.528
C00543=1101.652,429.870,400.454,-179.966,20.660,152.526
C00544=1101.646,429.624,400.495,-179.968,20.650,152.524
C00545=1101.640,429.377,400.536,-179.970,20.641,152.521
C00546=1101.635,429.132,400.577,-179.972,20.631,152.519
C00547=1101.629,428.884,400.618,-179.974,20.622,152.517
C00548=1101.622,428.638,400.658,-179.976,20.612,152.515
C00549=1101.617,428.392,400.700,-179.978,20.603,152.513
C00550=1101.612,428.146,400.740,-179.980,20.593,152.511
C00551=1101.606,427.899,400.782,-179.982,20.583,152.509
C00552=1101.600,427.653,400.822,-179.984,20.574,152.507
C00553=1101.594,427.406,400.863,-179.986,20.565,152.505
C00554=1101.588,427.160,400.904,-179.988,20.555,152.503
C00555=1101.582,426.913,400.945,-179.990,20.546,152.501
C00556=1101.576,426.666,400.986,-179.992,20.537,152.499
C00557=1101.570,426.420,401.026,-179.994,20.527,152.497
C00558=1101.564,426.173,401.067,-179.996,20.518,152.495
C00559=1101.558,425.927,401.108,-179.998,20.509,152.493
C00560=1101.552,425.680,401.148,-180.000,20.500,152.491
C00561=1101.546,425.433,401.189,179.997,20.490,152.489
C00562=1101.541,425.186,401.230,179.996,20.481,152.487
C00563=1101.534,424.886,401.279,179.994,20.470,152.485
C00564=1101.526,424.587,401.329,179.991,20.459,152.482
C00565=1101.519,424.287,401.377,179.989,20.448,152.480
C00566=1101.512,423.987,401.427,179.986,20.437,152.478
C00567=1101.506,423.699,401.474,179.983,20.427,152.476
C00568=1101.499,423.412,401.521,179.981,20.417,152.473
C00569=1101.493,423.165,401.561,179.979,20.407,152.471
C00570=1101.487,422.919,401.602,179.977,20.399,152.470
C00571=1101.481,422.672,401.643,179.974,20.389,152.468
C00572=1101.475,422.425,401.682,179.972,20.381,152.466
C00573=1101.470,422.179,401.723,179.970,20.372,152.464
C00574=1101.464,421.932,401.763,179.968,20.364,152.462
C00575=1101.457,421.685,401.803,179.966,20.355,152.460
C00576=1101.452,421.439,401.844,179.964,20.347,152.459
C00577=1101.445,421.192,401.884,179.962,20.338,152.457
C00578=1101.440,420.945,401.924,179.960,20.329,152.455
C00579=1101.434,420.699,401.964,179.958,20.321,152.453
C00580=1101.429,420.452,402.004,179.956,20.312,152.451
C00581=1101.422,420.206,402.045,179.954,20.304,152.450
C00582=1101.416,419.958,402.084,179.951,20.295,152.448
C00583=1101.411,419.712,402.124,179.949,20.287,152.446
C00584=1101.405,419.466,402.165,179.947,20.278,152.445
C00585=1101.399,419.218,402.205,179.945,20.270,152.443
C00586=1101.393,418.972,402.245,179.943,20.262,152.441
C00587=1101.388,418.725,402.284,179.941,20.253,152.439
C00588=1101.382,418.479,402.325,179.938,20.245,152.438
C00589=1101.376,418.232,402.365,179.936,20.237,152.436
C00590=1101.370,417.985,402.405,179.934,20.228,152.434
C00591=1101.364,417.739,402.444,179.932,20.220,152.433
C00592=1101.358,417.492,402.484,179.929,20.212,152.431
C00593=1101.353,417.245,402.525,179.927,20.204,152.429
C00594=1101.347,416.998,402.564,179.925,20.195,152.428
C00595=1101.341,416.751,402.603,179.923,20.187,152.426
C00596=1101.335,416.505,402.643,179.920,20.179,152.424
C00597=1101.330,416.258,402.683,179.918,20.171,152.423
C00598=1101.324,416.011,402.723,179.916,20.163,152.421
C00599=1101.318,415.764,402.763,179.914,20.156,152.420
C00600=1101.312,415.517,402.802,179.912,20.147,152.418
C00601=1101.306,415.271,402.842,179.910,20.139,152.416
C00602=1101.300,415.024,402.881,179.907,20.131,152.415
C00603=1101.294,414.777,402.921,179.905,20.123,152.413
C00604=1101.289,414.530,402.960,179.902,20.116,152.412
C00605=1101.282,414.284,403.000,179.901,20.108,152.410
C00606=1101.276,414.037,403.040,179.898,20.101,152.409
C00607=1101.271,413.790,403.079,179.896,20.093,152.407
C00608=1101.265,413.543,403.118,179.893,20.085,152.405
C00609=1101.258,413.297,403.158,179.891,20.077,152.404
C00610=1101.253,413.050,403.198,179.889,20.070,152.402
C00611=1101.247,412.803,403.237,179.887,20.062,152.401
C00612=1101.241,412.557,403.276,179.885,20.054,152.399
C00613=1101.235,412.309,403.315,179.882,20.046,152.398
C00614=1101.229,412.062,403.355,179.880,20.039,152.396
C00615=1101.224,411.816,403.394,179.878,20.031,152.395
C00616=1101.218,411.569,403.433,179.875,20.024,152.393
C00617=1101.213,411.354,403.468,179.873,20.017,152.392
C00618=1101.208,411.139,403.502,179.871,20.011,152.391
C00619=1101.203,410.923,403.536,179.869,20.004,152.390
C00620=1101.198,410.709,403.570,179.867,19.998,152.388
C00621=1101.193,410.493,403.604,179.865,19.991,152.387
C00622=1101.187,410.278,403.638,179.863,19.984,152.386
C00623=1101.183,410.063,403.673,179.861,19.978,152.384
C00624=1101.178,409.848,403.707,179.859,19.972,152.383
C00625=1101.172,409.602,403.746,179.857,19.965,152.382
C00626=1101.166,409.354,403.785,179.855,19.957,152.380
C00627=1101.161,409.108,403.824,179.852,19.950,152.379
C00628=1101.154,408.861,403.863,179.850,19.943,152.378
C00629=1101.149,408.614,403.903,179.848,19.935,152.376
C00630=1101.143,408.367,403.941,179.845,19.927,152.375
C00631=1101.138,408.120,403.980,179.843,19.921,152.373
C00632=1101.132,407.873,404.020,179.841,19.913,152.372
C00633=1101.126,407.627,404.059,179.839,19.906,152.370
C00634=1101.120,407.379,404.098,179.836,19.899,152.369
C00635=1101.114,407.133,404.136,179.833,19.892,152.368
C00636=1101.108,406.886,404.175,179.831,19.885,152.366
C00637=1101.103,406.639,404.214,179.829,19.878,152.365
C00638=1101.097,406.392,404.253,179.827,19.871,152.364
C00639=1101.091,406.145,404.292,179.824,19.864,152.362
C00640=1101.086,405.898,404.330,179.822,19.857,152.361
C00641=1101.079,405.651,404.369,179.819,19.850,152.360
C00642=1101.074,405.404,404.408,179.817,19.843,152.359
C00643=1101.068,405.157,404.447,179.815,19.836,152.357
C00644=1101.062,404.910,404.485,179.813,19.830,152.356
C00645=1101.057,404.664,404.524,179.810,19.823,152.355
C00646=1101.051,404.416,404.563,179.808,19.816,152.353
C00647=1101.045,404.170,404.601,179.805,19.809,152.352
C00648=1101.039,403.922,404.640,179.803,19.802,152.351
C00649=1101.033,403.676,404.678,179.800,19.795,152.350
C00650=1101.028,403.429,404.717,179.798,19.789,152.348
C00651=1101.022,403.182,404.756,179.795,19.782,152.347
C00652=1101.016,402.935,404.794,179.794,19.775,152.346
C00653=1101.010,402.687,404.833,179.791,19.768,152.345
C00654=1101.004,402.441,404.871,179.789,19.762,152.343
C00655=1100.999,402.194,404.910,179.786,19.755,152.342
C00656=1100.993,401.946,404.948,179.784,19.748,152.341
C00657=1100.987,401.700,404.987,179.781,19.742,152.340
C00658=1100.981,401.453,405.025,179.779,19.735,152.339
C00659=1100.975,401.206,405.063,179.776,19.729,152.337
C00660=1100.970,400.959,405.102,179.773,19.722,152.336
C00661=1100.964,400.713,405.140,179.772,19.715,152.335
C00662=1100.958,400.466,405.178,179.769,19.709,152.334
C00663=1100.952,400.218,405.216,179.766,19.702,152.333
C00664=1100.947,399.971,405.255,179.764,19.696,152.332
C00665=1100.941,399.724,405.293,179.762,19.690,152.330
C00666=1100.935,399.477,405.331,179.759,19.683,152.329
C00667=1100.929,399.230,405.370,179.757,19.677,152.328
C00668=1100.923,398.984,405.408,179.754,19.670,152.327
C00669=1100.918,398.737,405.446,179.752,19.664,152.326
C00670=1100.911,398.489,405.484,179.750,19.658,152.325
C00671=1100.906,398.242,405.522,179.747,19.652,152.323
C00672=1100.900,397.995,405.560,179.744,19.645,152.322
C00673=1100.895,397.780,405.593,179.743,19.640,152.321
C00674=1100.890,397.565,405.627,179.740,19.634,152.320
C00675=1100.885,397.350,405.660,179.738,19.629,152.320
C00676=1100.880,397.135,405.693,179.736,19.624,152.319
C00677=1100.875,396.920,405.725,179.734,19.618,152.318
C00678=1100.870,396.706,405.759,179.732,19.613,152.317
C00679=1100.865,396.490,405.792,179.729,19.608,152.316
C00680=1100.860,396.275,405.825,179.727,19.602,152.315
C00681=1100.854,396.028,405.863,179.725,19.596,152.314
C00682=1100.849,395.781,405.901,179.722,19.590,152.313
C00683=1100.843,395.534,405.939,179.720,19.584,152.312
C00684=1100.837,395.287,405.976,179.717,19.578,152.311
C00685=1100.831,395.039,406.014,179.714,19.572,152.310
C00686=1100.825,394.793,406.052,179.712,19.566,152.309
C00687=1100.820,394.545,406.090,179.710,19.560,152.307
C00688=1100.814,394.299,406.128,179.707,19.553,152.306
C00689=1100.808,394.052,406.165,179.704,19.548,152.305
C00690=1100.802,393.805,406.203,179.702,19.542,152.304
C00691=1100.796,393.558,406.240,179.700,19.536,152.303
C00692=1100.790,393.311,406.278,179.697,19.530,152.302
C00693=1100.785,393.063,406.317,179.694,19.524,152.301
C00694=1100.779,392.816,406.354,179.692,19.518,152.300
C00695=1100.773,392.569,406.392,179.689,19.512,152.299
C00696=1100.767,392.323,406.429,179.687,19.506,152.298
C00697=1100.762,392.075,406.466,179.684,19.501,152.298
C00698=1100.756,391.828,406.504,179.681,19.495,152.297
C00699=1100.750,391.582,406.542,179.679,19.489,152.296
C00700=1100.744,391.334,406.579,179.676,19.484,152.295
C00701=1100.738,391.088,406.617,179.674,19.478,152.294
C00702=1100.733,390.840,406.654,179.671,19.472,152.293
C00703=1100.727,390.593,406.691,179.669,19.467,152.292
C00704=1100.721,390.346,406.728,179.666,19.461,152.291
C00705=1100.715,390.099,406.766,179.663,19.455,152.290
C00706=1100.710,389.852,406.803,179.660,19.449,152.289
C00707=1100.704,389.605,406.841,179.658,19.444,152.288
C00708=1100.698,389.358,406.877,179.655,19.438,152.287
C00709=1100.692,389.111,406.915,179.653,19.433,152.286
C00710=1100.686,388.864,406.952,179.650,19.427,152.286
C00711=1100.680,388.617,406.990,179.648,19.422,152.285
C00712=1100.675,388.370,407.027,179.644,19.416,152.284
C00713=1100.669,388.123,407.065,179.642,19.410,152.283
C00714=1100.663,387.876,407.102,179.639,19.405,152.282
C00715=1100.657,387.628,407.139,179.636,19.399,152.281
C00716=1100.651,387.382,407.176,179.634,19.394,152.280
C00717=1100.645,387.135,407.213,179.631,19.388,152.279
C00718=1100.640,386.887,407.250,179.629,19.383,152.278
C00719=1100.634,386.641,407.288,179.626,19.377,152.278
C00720=1100.628,386.393,407.325,179.624,19.372,152.277
C00721=1100.623,386.146,407.362,179.621,19.367,152.276
C00722=1100.616,385.899,407.398,179.618,19.361,152.275
C00723=1100.611,385.652,407.435,179.615,19.356,152.274
C00724=1100.605,385.405,407.473,179.612,19.350,152.273
C00725=1100.600,385.158,407.510,179.610,19.345,152.273
C00726=1100.594,384.911,407.547,179.607,19.340,152.272
C00727=1100.588,384.664,407.583,179.604,19.334,152.271
C00728=1100.582,384.416,407.620,179.602,19.329,152.270
C00729=1100.572,383.999,407.683,179.598,19.320,152.269
C00730=1100.563,383.581,407.745,179.593,19.311,152.267
C00731=1100.553,383.163,407.808,179.588,19.303,152.266
C00732=1100.544,382.746,407.870,179.584,19.293,152.265
C00733=1100.538,382.499,407.906,179.581,19.288,152.264
C00734=1100.533,382.251,407.943,179.578,19.283,152.263
C00735=1100.526,382.004,407.980,179.575,19.278,152.262
C00736=1100.521,381.757,408.017,179.572,19.273,152.262
C00737=1100.514,381.510,408.053,179.570,19.268,152.261
C00738=1100.509,381.263,408.090,179.567,19.263,152.260
C00739=1100.503,381.016,408.127,179.564,19.257,152.259
C00740=1100.497,380.769,408.164,179.561,19.252,152.259
C00741=1100.491,380.521,408.199,179.559,19.248,152.258
C00742=1100.486,380.274,408.236,179.557,19.243,152.257
C00743=1100.481,380.027,408.273,179.554,19.238,152.256
C00744=1100.474,379.780,408.309,179.551,19.233,152.256
C00745=1100.469,379.533,408.346,179.548,19.228,152.255
C00746=1100.463,379.285,408.382,179.545,19.223,152.254
C00747=1100.457,379.038,408.419,179.542,19.218,152.254
C00748=1100.451,378.791,408.455,179.540,19.213,152.253
C00749=1100.445,378.544,408.492,179.537,19.208,152.252
C00750=1100.440,378.296,408.528,179.534,19.203,152.251
C00751=1100.433,378.049,408.565,179.531,19.198,152.251
C00752=1100.428,377.803,408.601,179.528,19.193,152.250
C00753=1100.422,377.555,408.637,179.525,19.188,152.249
C00754=1100.417,377.308,408.674,179.523,19.183,152.249
C00755=1100.411,377.061,408.710,179.520,19.179,152.248
C00756=1100.406,376.813,408.746,179.518,19.174,152.247
C00757=1100.399,376.566,408.783,179.515,19.169,152.247
C00758=1100.394,376.319,408.818,179.512,19.164,152.246
C00759=1100.388,376.072,408.855,179.509,19.159,152.245
C00760=1100.382,375.825,408.892,179.506,19.154,152.245
C00761=1100.377,375.578,408.928,179.503,19.149,152.244
C00762=1100.371,375.330,408.964,179.500,19.145,152.243
C00763=1100.365,375.083,409.000,179.498,19.140,152.243
C00764=1100.360,374.836,409.036,179.495,19.136,152.242
C00765=1100.354,374.588,409.072,179.492,19.131,152.241
C00766=1100.349,374.340,409.109,179.490,19.126,152.241
C00767=1100.343,374.094,409.145,179.486,19.121,152.240
C00768=1100.337,373.846,409.180,179.483,19.117,152.240
C00769=1100.331,373.599,409.217,179.480,19.112,152.239
C00770=1100.325,373.352,409.252,179.478,19.108,152.238
C00771=1100.320,373.104,409.288,179.475,19.103,152.238
C00772=1100.314,372.857,409.325,179.472,19.099,152.237
C00773=1100.308,372.610,409.360,179.469,19.094,152.237
C00774=1100.302,372.363,409.396,179.466,19.089,152.236
C00775=1100.296,372.116,409.432,179.464,19.085,152.235
C00776=1100.290,371.869,409.468,179.461,19.080,152.235
C00777=1100.285,371.621,409.504,179.458,19.076,152.234
C00778=1100.279,371.373,409.540,179.455,19.071,152.234
C00779=1100.273,371.127,409.576,179.452,19.067,152.233
C00780=1100.267,370.879,409.612,179.450,19.063,152.232
C00781=1100.258,370.489,409.668,179.445,19.055,152.232
C00782=1100.250,370.098,409.725,179.440,19.048,152.231
C00783=1100.241,369.707,409.781,179.436,19.041,152.230
C00784=1100.231,369.316,409.838,179.431,19.034,152.229
C00785=1100.225,369.069,409.873,179.429,19.030,152.228
C00786=1100.219,368.821,409.909,179.426,19.025,152.228
C00787=1100.214,368.574,409.944,179.422,19.021,152.227
C00788=1100.208,368.327,409.980,179.419,19.016,152.227
C00789=1100.203,368.080,410.015,179.417,19.012,152.226
C00790=1100.197,367.832,410.051,179.414,19.008,152.226
C00791=1100.191,367.585,410.086,179.411,19.003,152.225
C00792=1100.186,367.337,410.122,179.408,18.999,152.225
C00793=1100.180,367.090,410.158,179.406,18.995,152.224
C00794=1100.174,366.843,410.194,179.402,18.991,152.224
C00795=1100.169,366.596,410.229,179.399,18.986,152.223
C00796=1100.163,366.348,410.265,179.396,18.981,152.223
C00797=1100.157,366.101,410.300,179.394,18.978,152.222
C00798=1100.151,365.853,410.336,179.391,18.973,152.222
C00799=1100.146,365.606,410.370,179.387,18.969,152.221
C00800=1100.140,365.358,410.406,179.385,18.965,152.221
C00801=1100.134,365.111,410.441,179.382,18.961,152.220
C00802=1100.128,364.864,410.477,179.379,18.956,152.220
C00803=1100.123,364.617,410.512,179.375,18.952,152.219
C00804=1100.117,364.368,410.547,179.373,18.948,152.219
C00805=1100.111,364.121,410.582,179.370,18.944,152.218
C00806=1100.106,363.874,410.618,179.367,18.940,152.218
C00807=1100.099,363.627,410.653,179.364,18.936,152.217
C00808=1100.094,363.379,410.688,179.361,18.931,152.217
C00809=1100.088,363.132,410.723,179.358,18.927,152.216
C00810=1100.083,362.885,410.759,179.355,18.924,152.216
C00811=1100.077,362.637,410.794,179.352,18.920,152.216
C00812=1100.071,362.390,410.828,179.349,18.915,152.215
C00813=1100.065,362.142,410.864,179.347,18.911,152.215
C00814=1100.060,361.895,410.899,179.343,18.907,152.214
C00815=1100.054,361.648,410.934,179.340,18.903,152.214
C00816=1100.048,361.400,410.969,179.338,18.899,152.213
C00817=1100.042,361.153,411.004,179.334,18.895,152.213
C00818=1100.036,360.905,411.040,179.331,18.891,152.212
C00819=1100.031,360.657,411.074,179.329,18.887,152.212
C00820=1100.025,360.411,411.109,179.325,18.883,152.212
C00821=1100.019,360.162,411.144,179.323,18.879,152.211
C00822=1100.014,359.915,411.179,179.320,18.875,152.211
C00823=1100.007,359.667,411.214,179.316,18.871,152.210
C00824=1100.002,359.420,411.249,179.314,18.868,152.210
C00825=1099.997,359.173,411.284,179.310,18.863,152.210
C00826=1099.990,358.925,411.318,179.307,18.859,152.209
C00827=1099.985,358.678,411.354,179.305,18.856,152.209
C00828=1099.980,358.430,411.388,179.301,18.851,152.208
C00829=1099.973,358.182,411.423,179.299,18.848,152.208
C00830=1099.968,357.935,411.458,179.295,18.844,152.208
C00831=1099.962,357.688,411.492,179.292,18.840,152.207
C00832=1099.956,357.440,411.527,179.290,18.836,152.207
C00833=1099.947,357.064,411.580,179.285,18.830,152.206
C00834=1099.939,356.689,411.633,179.280,18.825,152.206
C00835=1099.930,356.314,411.685,179.276,18.819,152.205
C00836=1099.922,355.938,411.738,179.271,18.813,152.205
C00837=1099.915,355.690,411.772,179.268,18.809,152.204
C00838=1099.910,355.442,411.807,179.265,18.805,152.204
C00839=1099.905,355.195,411.842,179.262,18.802,152.204
C00840=1099.899,354.948,411.876,179.259,18.798,152.203
C00841=1099.893,354.700,411.911,179.256,18.794,152.203
C00842=1099.887,354.452,411.945,179.253,18.791,152.203
C00843=1099.882,354.205,411.980,179.250,18.787,152.202
C00844=1099.876,353.958,412.014,179.247,18.783,152.202
C00845=1099.870,353.710,412.049,179.244,18.779,152.202
C00846=1099.865,353.462,412.083,179.240,18.775,152.201
C00847=1099.859,353.215,412.117,179.238,18.772,152.201
C00848=1099.854,352.967,412.152,179.234,18.768,152.201
C00849=1099.847,352.719,412.186,179.232,18.765,152.200
C00850=1099.841,352.472,412.220,179.228,18.761,152.200
C00851=1099.836,352.224,412.255,179.226,18.758,152.200
C00852=1099.830,351.977,412.289,179.222,18.753,152.199
C00853=1099.824,351.729,412.324,179.220,18.750,152.199
C00854=1099.819,351.481,412.358,179.216,18.747,152.199
C00855=1099.813,351.234,412.392,179.213,18.743,152.199
C00856=1099.807,350.987,412.426,179.210,18.739,152.198
C00857=1099.802,350.739,412.461,179.207,18.736,152.198
C00858=1099.796,350.491,412.495,179.204,18.732,152.198
C00859=1099.790,350.243,412.529,179.201,18.729,152.197
C00860=1099.784,349.996,412.563,179.197,18.725,152.197
C00861=1099.779,349.748,412.597,179.195,18.722,152.197
C00862=1099.773,349.501,412.631,179.192,18.718,152.197
C00863=1099.767,349.254,412.666,179.189,18.715,152.196
C00864=1099.762,349.005,412.700,179.185,18.711,152.196
C00865=1099.756,348.758,412.734,179.183,18.708,152.196
C00866=1099.750,348.510,412.768,179.179,18.704,152.196
C00867=1099.744,348.263,412.802,179.176,18.701,152.195
C00868=1099.739,348.015,412.835,179.173,18.697,152.195
C00869=1099.734,347.768,412.870,179.170,18.694,152.195
C00870=1099.728,347.520,412.904,179.167,18.691,152.194
C00871=1099.722,347.272,412.937,179.164,18.687,152.194
C00872=1099.716,347.024,412.972,179.161,18.684,152.194
C00873=1099.710,346.777,413.006,179.158,18.680,152.194
C00874=1099.704,346.529,413.039,179.155,18.677,152.193
C00875=1099.699,346.282,413.074,179.151,18.673,152.193
C00876=1099.694,346.034,413.107,179.149,18.670,152.193
C00877=1099.688,345.787,413.141,179.145,18.666,152.193
C00878=1099.682,345.539,413.175,179.142,18.663,152.193
C00879=1099.676,345.291,413.209,179.139,18.659,152.192
C00880=1099.671,345.044,413.243,179.136,18.656,152.192
C00881=1099.665,344.796,413.276,179.133,18.653,152.192
C00882=1099.659,344.549,413.310,179.129,18.650,152.192
C00883=1099.654,344.301,413.343,179.127,18.646,152.191
C00884=1099.647,344.053,413.378,179.123,18.643,152.191
C00885=1099.639,343.679,413.428,179.119,18.638,152.191
C00886=1099.630,343.306,413.479,179.114,18.633,152.191
C00887=1099.621,342.933,413.530,179.110,18.628,152.190
C00888=1099.613,342.559,413.580,179.105,18.623,152.190
C00889=1099.607,342.311,413.614,179.101,18.620,152.190
C00890=1099.602,342.064,413.648,179.098,18.617,152.190
C00891=1099.596,341.816,413.681,179.095,18.614,152.189
C00892=1099.590,341.568,413.714,179.092,18.610,152.189
C00893=1099.585,341.321,413.748,179.089,18.607,152.189
C00894=1099.579,341.073,413.782,179.086,18.604,152.189
C00895=1099.573,340.825,413.815,179.082,18.601,152.189
C00896=1099.567,340.578,413.849,179.080,18.597,152.188
C00897=1099.561,340.330,413.882,179.076,18.594,152.188
C00898=1099.556,340.082,413.915,179.073,18.591,152.188
C00899=1099.550,339.834,413.949,179.070,18.588,152.188
C00900=1099.545,339.586,413.982,179.067,18.584,152.188
C00901=1099.539,339.340,414.016,179.064,18.582,152.188
C00902=1099.534,339.092,414.049,179.061,18.578,152.187
C00903=1099.528,338.844,414.082,179.057,18.575,152.187
C00904=1099.522,338.596,414.115,179.054,18.572,152.187
C00905=1099.516,338.348,414.148,179.051,18.569,152.187
C00906=1099.511,338.101,414.182,179.048,18.566,152.187
C00907=1099.505,337.853,414.215,179.045,18.563,152.187
C00908=1099.499,337.605,414.248,179.042,18.560,152.186
C00909=1099.494,337.357,414.281,179.038,18.556,152.186
C00910=1099.488,337.109,414.314,179.035,18.554,152.186
C00911=1099.482,336.861,414.348,179.032,18.551,152.186
C00912=1099.476,336.614,414.381,179.029,18.547,152.186
C00913=1099.471,336.366,414.414,179.026,18.544,152.186
C00914=1099.465,336.118,414.447,179.023,18.542,152.186
C00915=1099.459,335.871,414.480,179.019,18.538,152.186
C00916=1099.454,335.623,414.513,179.016,18.535,152.185
C00917=1099.448,335.375,414.546,179.013,18.533,152.185
C00918=1099.442,335.128,414.579,179.010,18.529,152.185
C00919=1099.436,334.880,414.612,179.007,18.526,152.185
C00920=1099.431,334.632,414.646,179.004,18.523,152.185
C00921=1099.425,334.384,414.678,179.001,18.521,152.185
C00922=1099.420,334.137,414.711,178.997,18.517,152.185
C00923=1099.414,333.889,414.744,178.994,18.514,152.185
C00924=1099.408,333.641,414.777,178.991,18.512,152.185
C00925=1099.402,333.393,414.810,178.988,18.509,152.184
C00926=1099.396,333.145,414.843,178.984,18.505,152.184
C00927=1099.391,332.898,414.876,178.981,18.503,152.184
C00928=1099.386,332.650,414.908,178.978,18.500,152.184
C00929=1099.380,332.402,414.941,178.975,18.497,152.184
C00930=1099.374,332.154,414.975,178.972,18.494,152.184
C00931=1099.368,331.907,415.007,178.969,18.491,152.184
C00932=1099.363,331.658,415.040,178.966,18.488,152.184
C00933=1099.356,331.411,415.073,178.963,18.485,152.184
C00934=1099.351,331.164,415.105,178.959,18.482,152.183
C00935=1099.345,330.915,415.138,178.956,18.480,152.184
C00936=1099.339,330.668,415.170,178.953,18.477,152.183
C00937=1099.330,330.288,415.220,178.947,18.472,152.183
C00938=1099.321,329.908,415.271,178.943,18.468,152.183
C00939=1099.313,329.529,415.320,178.937,18.464,152.183
C00940=1099.304,329.149,415.370,178.933,18.460,152.183
C00941=1099.297,328.902,415.403,178.930,18.457,152.183
C00942=1099.293,328.654,415.435,178.927,18.454,152.183
C00943=1099.286,328.406,415.468,178.923,18.451,152.183
C00944=1099.280,328.158,415.500,178.920,18.449,152.183
C00945=1099.275,327.910,415.533,178.917,18.446,152.183
C00946=1099.270,327.663,415.565,178.914,18.444,152.183
C00947=1099.263,327.415,415.598,178.910,18.440,152.183
C00948=1099.257,327.167,415.630,178.907,18.438,152.183
C00949=1099.252,326.919,415.663,178.904,18.435,152.183
C00950=1099.246,326.671,415.695,178.901,18.432,152.183
C00951=1099.240,326.423,415.727,178.898,18.430,152.182
C00952=1099.235,326.175,415.760,178.895,18.427,152.183
C00953=1099.229,325.927,415.792,178.891,18.424,152.182
C00954=1099.223,325.680,415.824,178.888,18.422,152.182
C00955=1099.217,325.432,415.856,178.885,18.419,152.182
C00956=1099.212,325.183,415.889,178.881,18.416,152.182
C00957=1099.206,324.936,415.921,178.879,18.414,152.182
C00958=1099.200,324.688,415.953,178.875,18.410,152.182
C00959=1099.194,324.440,415.985,178.872,18.408,152.182
C00960=1099.189,324.193,416.017,178.869,18.405,152.182
C00961=1099.184,323.944,416.050,178.865,18.403,152.182
C00962=1099.178,323.697,416.082,178.862,18.400,152.182
C00963=1099.172,323.449,416.114,178.859,18.398,152.182
C00964=1099.166,323.201,416.146,178.856,18.395,152.182
C00965=1099.161,322.953,416.178,178.852,18.392,152.182
C00966=1099.155,322.705,416.210,178.849,18.389,152.182
C00967=1099.150,322.458,416.243,178.846,18.387,152.182
C00968=1099.144,322.210,416.275,178.843,18.385,152.182
C00969=1099.138,321.961,416.307,178.840,18.382,152.182
C00970=1099.132,321.714,416.339,178.837,18.379,152.182
C00971=1099.126,321.466,416.371,178.834,18.377,152.182
C00972=1099.121,321.218,416.402,178.830,18.374,152.182
C00973=1099.116,320.970,416.435,178.827,18.371,152.182
C00974=1099.110,320.722,416.466,178.823,18.369,152.182
C00975=1099.104,320.474,416.498,178.820,18.366,152.182
C00976=1099.099,320.226,416.530,178.817,18.363,152.182
C00977=1099.093,319.978,416.562,178.814,18.361,152.182
C00978=1099.087,319.731,416.594,178.811,18.358,152.182
C00979=1099.081,319.482,416.626,178.807,18.355,152.182
C00980=1099.076,319.235,416.658,178.804,18.353,152.182
C00981=1099.070,318.987,416.690,178.801,18.350,152.182
C00982=1099.065,318.739,416.721,178.798,18.348,152.182
C00983=1099.059,318.491,416.754,178.794,18.346,152.182
C00984=1099.054,318.243,416.786,178.791,18.343,152.182
C00985=1099.048,317.995,416.818,178.788,18.340,152.182
C00986=1099.043,317.747,416.849,178.785,18.338,152.182
C00987=1099.037,317.499,416.881,178.782,18.335,152.182
C00988=1099.032,317.251,416.912,178.778,18.332,152.182
C00989=1099.023,316.865,416.962,178.773,18.329,152.182
C00990=1099.014,316.478,417.011,178.769,18.325,152.182
C00991=1099.006,316.092,417.061,178.763,18.321,152.182
C00992=1098.997,315.705,417.110,178.758,18.317,152.182
C00993=1098.991,315.457,417.142,178.755,18.314,152.182
C00994=1098.986,315.210,417.173,178.752,18.312,152.182
C00995=1098.979,314.962,417.205,178.749,18.310,152.182
C00996=1098.974,314.714,417.236,178.745,18.307,152.182
C00997=1098.968,314.466,417.268,178.742,18.305,152.182
C00998=1098.962,314.218,417.299,178.739,18.303,152.182
C00999=1098.956,313.970,417.330,178.735,18.300,152.182
C01000=1098.951,313.722,417.362,178.732,18.297,152.182
C01001=1098.945,313.474,417.394,178.728,18.296,152.183
C01002=1098.939,313.226,417.424,178.725,18.293,152.183
C01003=1098.934,312.979,417.456,178.722,18.291,152.183
C01004=1098.928,312.730,417.487,178.719,18.289,152.183
C01005=1098.922,312.482,417.518,178.715,18.286,152.183
C01006=1098.916,312.234,417.550,178.712,18.284,152.183
C01007=1098.910,311.986,417.580,178.709,18.281,152.183
C01008=1098.904,311.738,417.613,178.706,18.279,152.183
C01009=1098.899,311.490,417.643,178.702,18.277,152.183
C01010=1098.893,311.243,417.675,178.699,18.275,152.183
C01011=1098.887,310.994,417.706,178.696,18.273,152.183
C01012=1098.882,310.747,417.738,178.693,18.270,152.183
C01013=1098.876,310.499,417.768,178.689,18.268,152.183
C01014=1098.870,310.251,417.800,178.686,18.266,152.184
C01015=1098.864,310.003,417.830,178.683,18.263,152.184
C01016=1098.859,309.755,417.862,178.679,18.261,152.184
C01017=1098.852,309.507,417.893,178.676,18.259,152.184
C01018=1098.847,309.259,417.924,178.673,18.257,152.184
C01019=1098.842,309.011,417.955,178.670,18.254,152.184
C01020=1098.836,308.762,417.986,178.667,18.252,152.184
C01021=1098.830,308.515,418.018,178.663,18.250,152.184
C01022=1098.824,308.267,418.048,178.660,18.248,152.184
C01023=1098.819,308.019,418.079,178.657,18.245,152.184
C01024=1098.813,307.771,418.110,178.653,18.243,152.184
C01025=1098.807,307.523,418.141,178.650,18.241,152.185
C01026=1098.802,307.275,418.172,178.647,18.239,152.185
C01027=1098.796,307.028,418.203,178.643,18.236,152.185
C01028=1098.790,306.779,418.234,178.640,18.234,152.185
C01029=1098.785,306.531,418.265,178.637,18.232,152.185
C01030=1098.779,306.283,418.295,178.634,18.230,152.185
C01031=1098.774,306.036,418.327,178.630,18.227,152.185
C01032=1098.767,305.787,418.358,178.627,18.225,152.185
C01033=1098.762,305.539,418.389,178.624,18.223,152.185
C01034=1098.756,305.291,418.419,178.620,18.221,152.185
C01035=1098.751,305.043,418.450,178.616,18.218,152.186
C01036=1098.745,304.796,418.481,178.613,18.216,152.186
C01037=1098.740,304.548,418.512,178.610,18.214,152.186
C01038=1098.734,304.299,418.543,178.606,18.211,152.186
C01039=1098.728,304.051,418.573,178.604,18.210,152.186
C01040=1098.723,303.803,418.604,178.601,18.208,152.186
C01041=1098.714,303.419,418.652,178.595,18.203,152.186
C01042=1098.705,303.035,418.699,178.590,18.200,152.186
C01043=1098.696,302.651,418.746,178.585,18.197,152.187
C01044=1098.688,302.268,418.794,178.580,18.194,152.187
C01045=1098.682,302.020,418.824,178.577,18.191,152.187
C01046=1098.677,301.771,418.855,178.573,18.190,152.187
C01047=1098.671,301.524,418.886,178.570,18.187,152.187
C01048=1098.665,301.276,418.916,178.566,18.185,152.187
C01049=1098.660,301.028,418.947,178.563,18.183,152.187
C01050=1098.654,300.780,418.977,178.560,18.181,152.187
C01051=1098.649,300.532,419.008,178.557,18.179,152.188
C01052=1098.643,300.283,419.038,178.553,18.176,152.188
C01053=1098.638,300.035,419.068,178.550,18.174,152.188
C01054=1098.633,299.787,419.099,178.547,18.172,152.188
C01055=1098.627,299.539,419.130,178.543,18.170,152.188
C01056=1098.621,299.292,419.160,178.540,18.168,152.188
C01057=1098.615,299.044,419.190,178.537,18.165,152.188
C01058=1098.610,298.795,419.220,178.533,18.164,152.189
C01059=1098.605,298.547,419.251,178.530,18.161,152.189
C01060=1098.599,298.299,419.281,178.527,18.159,152.189
C01061=1098.594,298.051,419.312,178.524,18.158,152.189
C01062=1098.588,297.803,419.342,178.521,18.156,152.189
C01063=1098.582,297.555,419.372,178.517,18.153,152.189
C01064=1098.576,297.307,419.402,178.514,18.151,152.189
C01065=1098.571,297.059,419.433,178.511,18.149,152.189
C01066=1098.565,296.811,419.462,178.507,18.147,152.190
C01067=1098.559,296.563,419.493,178.504,18.145,152.190
C01068=1098.554,296.315,419.523,178.500,18.143,152.190
C01069=1098.548,296.067,419.553,178.497,18.141,152.190
C01070=1098.542,295.819,419.583,178.494,18.139,152.190
C01071=1098.537,295.571,419.614,178.490,18.137,152.190
C01072=1098.532,295.322,419.644,178.487,18.135,152.191
C01073=1098.526,295.075,419.674,178.483,18.133,152.191
C01074=1098.520,294.826,419.704,178.481,18.131,152.191
C01075=1098.514,294.578,419.734,178.477,18.129,152.191
C01076=1098.509,294.330,419.764,178.474,18.127,152.191
C01077=1098.503,294.082,419.794,178.471,18.125,152.191
C01078=1098.497,293.834,419.824,178.467,18.123,152.192
C01079=1098.492,293.586,419.854,178.464,18.121,152.192
C01080=1098.486,293.338,419.884,178.461,18.119,152.192
C01081=1098.480,293.090,419.914,178.457,18.117,152.192
C01082=1098.475,292.842,419.944,178.454,18.115,152.192
C01083=1098.468,292.594,419.973,178.451,18.114,152.193
C01084=1098.463,292.346,420.004,178.448,18.111,152.193
C01085=1098.457,292.097,420.033,178.444,18.109,152.193
C01086=1098.452,291.849,420.063,178.441,18.108,152.193
C01087=1098.446,291.601,420.093,178.437,18.106,152.193
C01088=1098.440,291.353,420.123,178.434,18.103,152.193
C01089=1098.435,291.104,420.153,178.430,18.101,152.194
C01090=1098.429,290.856,420.183,178.427,18.099,152.194
C01091=1098.423,290.608,420.213,178.424,18.098,152.194
C01092=1098.418,290.361,420.243,178.421,18.096,152.194
C01093=1098.410,289.990,420.287,178.416,18.093,152.194
C01094=1098.401,289.620,420.331,178.411,18.090,152.195
C01095=1098.392,289.250,420.375,178.406,18.087,152.195
C01096=1098.384,288.880,420.419,178.401,18.085,152.195
C01097=1098.378,288.632,420.449,178.397,18.083,152.196
C01098=1098.373,288.384,420.478,178.394,18.081,152.196
C01099=1098.367,288.135,420.508,178.391,18.079,152.196
C01100=1098.361,287.888,420.538,178.387,18.077,152.196
C01101=1098.355,287.639,420.567,178.384,18.075,152.196
C01102=1098.350,287.391,420.597,178.381,18.074,152.197
C01103=1098.344,287.143,420.626,178.378,18.072,152.197
C01104=1098.338,286.895,420.655,178.374,18.070,152.197
C01105=1098.333,286.646,420.685,178.371,18.068,152.197
C01106=1098.327,286.399,420.715,178.367,18.066,152.197
C01107=1098.321,286.150,420.744,178.364,18.064,152.198
C01108=1098.315,285.902,420.774,178.361,18.063,152.198
C01109=1098.310,285.654,420.803,178.358,18.061,152.198
C01110=1098.304,285.406,420.832,178.354,18.059,152.198
C01111=1098.299,285.158,420.862,178.351,18.057,152.198
C01112=1098.293,284.909,420.892,178.347,18.055,152.199
C01113=1098.287,284.661,420.921,178.344,18.053,152.199
C01114=1098.282,284.413,420.950,178.341,18.052,152.199
C01115=1098.277,284.165,420.980,178.338,18.050,152.199
C01116=1098.270,283.917,421.009,178.334,18.048,152.199
C01117=1098.265,283.668,421.038,178.331,18.046,152.200
C01118=1098.259,283.421,421.067,178.327,18.044,152.200
C01119=1098.254,283.172,421.097,178.325,18.043,152.200
C01120=1098.248,282.924,421.126,178.321,18.041,152.200
C01121=1098.242,282.675,421.155,178.318,18.039,152.201
C01122=1098.237,282.428,421.184,178.314,18.037,152.201
C01123=1098.232,282.179,421.213,178.311,18.035,152.201
C01124=1098.225,281.931,421.242,178.307,18.033,152.201
C01125=1098.220,281.683,421.272,178.304,18.032,152.201
C01126=1098.214,281.435,421.301,178.301,18.030,152.202
C01127=1098.209,281.186,421.330,178.297,18.028,152.202
C01128=1098.203,280.938,421.359,178.294,18.026,152.202
C01129=1098.198,280.690,421.388,178.291,18.025,152.202
C01130=1098.192,280.442,421.417,178.288,18.023,152.203
C01131=1098.186,280.194,421.447,178.284,18.021,152.203
C01132=1098.180,279.945,421.475,178.281,18.020,152.203
C01133=1098.175,279.697,421.504,178.277,18.018,152.203
C01134=1098.169,279.449,421.533,178.274,18.016,152.204
C01135=1098.163,279.200,421.562,178.271,18.014,152.204
C01136=1098.158,278.952,421.591,178.267,18.013,152.204
C01137=1098.152,278.704,421.620,178.264,18.011,152.204
C01138=1098.147,278.455,421.649,178.260,18.009,152.205
C01139=1098.141,278.208,421.678,178.258,18.007,152.205
C01140=1098.135,277.960,421.707,178.254,18.006,152.205
C01141=1098.130,277.711,421.735,178.250,18.004,152.205
C01142=1098.124,277.463,421.764,178.247,18.002,152.206
C01143=1098.119,277.215,421.794,178.244,18.001,152.206
C01144=1098.113,276.966,421.822,178.241,17.999,152.206
C01145=1098.105,276.605,421.864,178.235,17.996,152.206
C01146=1098.096,276.245,421.905,178.231,17.994,152.207
C01147=1098.088,275.884,421.947,178.226,17.991,152.207
C01148=1098.080,275.524,421.990,178.221,17.989,152.207
C01149=1098.074,275.275,422.018,178.218,17.987,152.208
C01150=1098.068,275.027,422.046,178.215,17.986,152.208
C01151=1098.063,274.779,422.075,178.212,17.984,152.208
C01152=1098.058,274.530,422.104,178.208,17.983,152.209
C01153=1098.052,274.283,422.133,178.204,17.981,152.209
C01154=1098.046,274.034,422.161,178.202,17.979,152.209
C01155=1098.040,273.786,422.190,178.198,17.978,152.209
C01156=1098.035,273.537,422.218,178.195,17.976,152.209
C01157=1098.029,273.289,422.247,178.191,17.974,152.210
C01158=1098.024,273.041,422.275,178.188,17.973,152.210
C01159=1098.018,272.793,422.304,178.185,17.971,152.210
C01160=1098.012,272.544,422.332,178.181,17.969,152.210
C01161=1098.007,272.296,422.361,178.177,17.968,152.211
C01162=1098.001,272.047,422.390,178.175,17.966,152.211
C01163=1097.995,271.799,422.418,178.171,17.964,152.211
C01164=1097.989,271.551,422.447,178.168,17.963,152.212
C01165=1097.984,271.303,422.475,178.164,17.961,152.212
C01166=1097.978,271.054,422.503,178.161,17.960,152.212
C01167=1097.973,270.806,422.531,178.158,17.958,152.212
C01168=1097.967,270.558,422.561,178.154,17.956,152.213
C01169=1097.962,270.310,422.588,178.151,17.955,152.213
C01170=1097.956,270.061,422.617,178.148,17.953,152.213
C01171=1097.950,269.813,422.645,178.144,17.951,152.213
C01172=1097.944,269.564,422.673,178.141,17.950,152.214
C01173=1097.939,269.315,422.701,178.138,17.949,152.214
C01174=1097.933,269.068,422.730,178.134,17.947,152.214
C01175=1097.927,268.819,422.758,178.131,17.945,152.215
C01176=1097.922,268.571,422.786,178.128,17.944,152.215
C01177=1097.916,268.322,422.815,178.124,17.942,152.215
C01178=1097.910,268.074,422.843,178.121,17.941,152.215
C01179=1097.905,267.826,422.871,178.117,17.939,152.216
C01180=1097.899,267.578,422.899,178.114,17.938,152.216
C01181=1097.894,267.330,422.927,178.111,17.936,152.216
C01182=1097.888,267.081,422.955,178.107,17.934,152.217
C01183=1097.882,266.833,422.983,178.104,17.933,152.217
C01184=1097.876,266.584,423.012,178.101,17.931,152.217
C01185=1097.871,266.336,423.039,178.097,17.929,152.217
C01186=1097.865,266.087,423.068,178.094,17.929,152.218
C01187=1097.860,265.839,423.096,178.091,17.927,152.218
C01188=1097.854,265.590,423.124,178.088,17.925,152.218
C01189=1097.849,265.342,423.152,178.085,17.924,152.219
C01190=1097.843,265.094,423.180,178.081,17.922,152.219
C01191=1097.837,264.846,423.208,178.077,17.921,152.219
C01192=1097.832,264.598,423.236,178.074,17.919,152.219
C01193=1097.825,264.349,423.264,178.071,17.917,152.220
C01194=1097.820,264.100,423.291,178.067,17.916,152.220
C01195=1097.814,263.852,423.320,178.064,17.914,152.220
C01196=1097.809,263.604,423.348,178.061,17.913,152.221
C01197=1097.800,263.246,423.387,178.056,17.911,152.221
C01198=1097.792,262.888,423.428,178.051,17.908,152.221
C01199=1097.784,262.530,423.468,178.046,17.907,152.222
C01200=1097.775,262.172,423.508,178.042,17.905,152.222
C01201=1097.770,261.924,423.535,178.038,17.903,152.223
C01202=1097.764,261.676,423.563,178.034,17.902,152.223
C01203=1097.758,261.427,423.591,178.032,17.900,152.223
C01204=1097.752,261.179,423.619,178.028,17.899,152.224
C01205=1097.747,260.930,423.646,178.024,17.897,152.224
C01206=1097.741,260.682,423.674,178.021,17.896,152.224
C01207=1097.735,260.434,423.702,178.018,17.895,152.225
C01208=1097.730,260.185,423.729,178.014,17.893,152.225
C01209=1097.724,259.936,423.757,178.011,17.892,152.225
C01210=1097.718,259.689,423.785,178.008,17.890,152.225
C01211=1097.713,259.439,423.812,178.005,17.889,152.226
C01212=1097.707,259.191,423.840,178.001,17.887,152.226
C01213=1097.701,258.944,423.867,177.998,17.886,152.226
C01214=1097.696,258.694,423.895,177.995,17.884,152.227
C01215=1097.689,258.446,423.922,177.991,17.883,152.227
C01216=1097.684,258.198,423.950,177.987,17.882,152.227
C01217=1097.678,257.949,423.978,177.985,17.880,152.228
C01218=1097.673,257.701,424.005,177.981,17.879,152.228
C01219=1097.667,257.453,424.033,177.977,17.877,152.228
C01220=1097.661,257.204,424.060,177.974,17.876,152.229
C01221=1097.656,256.956,424.088,177.971,17.874,152.229
C01222=1097.651,256.707,424.115,177.968,17.873,152.229
C01223=1097.645,256.459,424.142,177.964,17.871,152.230
C01224=1097.639,256.210,424.170,177.961,17.870,152.230
C01225=1097.633,255.962,424.197,177.958,17.869,152.230
C01226=1097.628,255.713,424.224,177.954,17.867,152.231
C01227=1097.622,255.465,424.251,177.951,17.866,152.231
C01228=1097.616,255.216,424.279,177.948,17.865,152.231
C01229=1097.610,254.968,424.306,177.944,17.863,152.232
C01230=1097.605,254.720,424.334,177.941,17.862,152.232
C01231=1097.600,254.471,424.361,177.938,17.860,152.232
C01232=1097.594,254.222,424.388,177.934,17.858,152.232
C01233=1097.588,253.974,424.416,177.931,17.858,152.233
C01234=1097.582,253.726,424.443,177.928,17.856,152.233
C01235=1097.577,253.477,424.470,177.924,17.854,152.233
C01236=1097.572,253.229,424.497,177.921,17.853,152.234
C01237=1097.566,252.981,424.525,177.917,17.852,152.234
C01238=1097.560,252.731,424.552,177.914,17.851,152.234
C01239=1097.555,252.483,424.579,177.911,17.849,152.235
C01240=1097.549,252.234,424.606,177.907,17.847,152.235
C01241=1097.543,251.987,424.633,177.905,17.846,152.235
C01242=1097.538,251.738,424.660,177.901,17.845,152.236
C01243=1097.532,251.490,424.687,177.898,17.843,152.236
C01244=1097.527,251.241,424.714,177.894,17.842,152.236
C01245=1097.521,250.992,424.741,177.891,17.840,152.237
C01246=1097.516,250.743,424.768,177.888,17.839,152.237
C01247=1097.510,250.496,424.796,177.884,17.838,152.237
C01248=1097.505,250.247,424.823,177.881,17.836,152.238
C01249=1097.496,249.886,424.862,177.876,17.834,152.238
C01250=1097.488,249.525,424.901,177.871,17.832,152.239
C01251=1097.480,249.165,424.940,177.867,17.830,152.239
C01252=1097.472,248.803,424.979,177.862,17.828,152.239
C01253=1097.467,248.555,425.006,177.858,17.827,152.240
C01254=1097.461,248.307,425.033,177.856,17.826,152.240
C01255=1097.456,248.058,425.060,177.852,17.824,152.240
C01256=1097.450,247.810,425.087,177.848,17.822,152.241
C01257=1097.445,247.561,425.114,177.845,17.821,152.241
C01258=1097.439,247.313,425.140,177.842,17.819,152.241
C01259=1097.434,247.064,425.167,177.839,17.819,152.242
C01260=1097.428,246.816,425.194,177.835,17.817,152.242
C01261=1097.423,246.567,425.221,177.832,17.816,152.242
C01262=1097.417,246.319,425.248,177.829,17.814,152.243
C01263=1097.411,246.071,425.274,177.826,17.814,152.243
C01264=1097.405,245.821,425.301,177.822,17.812,152.243
C01265=1097.400,245.572,425.328,177.819,17.810,152.244
C01266=1097.394,245.324,425.354,177.816,17.809,152.244
C01267=1097.389,245.075,425.381,177.812,17.808,152.244
C01268=1097.383,244.827,425.408,177.809,17.807,152.245
C01269=1097.377,244.579,425.434,177.805,17.805,152.245
C01270=1097.371,244.330,425.461,177.803,17.804,152.245
C01271=1097.366,244.081,425.488,177.799,17.803,152.246
C01272=1097.361,243.833,425.514,177.796,17.802,152.246
C01273=1097.355,243.584,425.541,177.792,17.800,152.246
C01274=1097.349,243.336,425.568,177.789,17.798,152.247
C01275=1097.344,243.087,425.593,177.786,17.798,152.247
C01276=1097.338,242.839,425.620,177.782,17.796,152.247
C01277=1097.332,242.590,425.647,177.779,17.795,152.248
C01278=1097.326,242.342,425.673,177.775,17.793,152.248
C01279=1097.321,242.093,425.699,177.773,17.793,152.248
C01280=1097.315,241.845,425.726,177.769,17.791,152.249
C01281=1097.309,241.596,425.753,177.766,17.790,152.249
C01282=1097.304,241.347,425.779,177.762,17.788,152.250
C01283=1097.298,241.099,425.805,177.759,17.788,152.250
C01284=1097.292,240.851,425.832,177.756,17.786,152.250
C01285=1097.287,240.602,425.858,177.753,17.785,152.251
C01286=1097.282,240.354,425.884,177.749,17.783,152.251
C01287=1097.276,240.105,425.910,177.746,17.783,152.251
C01288=1097.270,239.857,425.937,177.743,17.781,152.252
C01289=1097.265,239.608,425.963,177.740,17.780,152.252
C01290=1097.259,239.359,425.989,177.736,17.778,152.252
C01291=1097.253,239.111,426.016,177.732,17.777,152.253
C01292=1097.248,238.862,426.042,177.729,17.776,152.253
C01293=1097.242,238.614,426.068,177.726,17.774,152.253
C01294=1097.237,238.365,426.094,177.723,17.773,152.254
C01295=1097.231,238.116,426.121,177.719,17.772,152.254
C01296=1097.225,237.867,426.147,177.716,17.771,152.254
C01297=1097.220,237.619,426.174,177.713,17.769,152.255
C01298=1097.213,237.370,426.199,177.710,17.769,152.255
C01299=1097.208,237.123,426.225,177.706,17.767,152.256
C01300=1097.203,236.874,426.251,177.703,17.766,152.256
C01301=1097.195,236.505,426.290,177.698,17.764,152.256
C01302=1097.186,236.138,426.329,177.693,17.763,152.257
C01303=1097.178,235.770,426.367,177.688,17.760,152.257
C01304=1097.169,235.402,426.406,177.683,17.759,152.258
C01305=1097.165,235.154,426.432,177.680,17.757,152.258
C01306=1097.159,234.905,426.458,177.677,17.756,152.259
C01307=1097.153,234.657,426.484,177.674,17.755,152.259
C01308=1097.147,234.408,426.510,177.670,17.754,152.259
C01309=1097.142,234.159,426.536,177.667,17.752,152.260
C01310=1097.137,233.911,426.561,177.664,17.751,152.260
C01311=1097.131,233.662,426.588,177.661,17.750,152.260
C01312=1097.125,233.414,426.613,177.657,17.749,152.261
C01313=1097.119,233.165,426.639,177.654,17.748,152.261
C01314=1097.114,232.916,426.665,177.650,17.746,152.261
C01315=1097.109,232.668,426.691,177.647,17.745,152.262
C01316=1097.102,232.419,426.717,177.644,17.744,152.262
C01317=1097.097,232.170,426.743,177.641,17.743,152.263
C01318=1097.092,231.921,426.768,177.638,17.742,152.263
C01319=1097.085,231.673,426.794,177.634,17.740,152.263
C01320=1097.080,231.425,426.819,177.631,17.739,152.264
C01321=1097.075,231.176,426.846,177.627,17.738,152.264
C01322=1097.068,230.928,426.871,177.624,17.737,152.264
C01323=1097.063,230.679,426.897,177.621,17.735,152.265
C01324=1097.058,230.430,426.923,177.618,17.734,152.265
C01325=1097.052,230.182,426.948,177.614,17.733,152.265
C01326=1097.046,229.933,426.974,177.611,17.732,152.266
C01327=1097.040,229.684,426.999,177.608,17.731,152.266
C01328=1097.035,229.436,427.025,177.605,17.730,152.267
C01329=1097.030,229.187,427.051,177.601,17.728,152.267
C01330=1097.024,228.938,427.076,177.598,17.727,152.267
C01331=1097.018,228.689,427.102,177.595,17.726,152.268
C01332=1097.013,228.441,427.127,177.591,17.725,152.268
C01333=1097.007,228.192,427.153,177.588,17.724,152.268
C01334=1097.001,227.943,427.178,177.585,17.723,152.269
C01335=1096.996,227.694,427.204,177.582,17.722,152.269
C01336=1096.990,227.446,427.229,177.578,17.720,152.270
C01337=1096.984,227.197,427.255,177.575,17.719,152.270
C01338=1096.978,226.949,427.281,177.572,17.718,152.270
C01339=1096.973,226.701,427.306,177.568,17.717,152.271
C01340=1096.967,226.452,427.332,177.566,17.716,152.271
C01341=1096.962,226.203,427.357,177.562,17.715,152.272
C01342=1096.956,225.954,427.382,177.559,17.714,152.272
C01343=1096.951,225.705,427.408,177.555,17.712,152.272
C01344=1096.945,225.457,427.433,177.552,17.711,152.273
C01345=1096.940,225.208,427.459,177.549,17.710,152.273
C01346=1096.934,224.960,427.484,177.546,17.709,152.273
C01347=1096.927,224.711,427.509,177.543,17.708,152.274
C01348=1096.923,224.462,427.534,177.539,17.707,152.274
C01349=1096.917,224.213,427.559,177.536,17.705,152.274
C01350=1096.912,223.965,427.585,177.532,17.704,152.275
C01351=1096.906,223.717,427.610,177.529,17.703,152.275
C01352=1096.900,223.467,427.636,177.526,17.702,152.276
C01353=1096.892,223.091,427.674,177.521,17.700,152.276
C01354=1096.883,222.715,427.712,177.516,17.698,152.277
C01355=1096.875,222.339,427.750,177.511,17.697,152.277
C01356=1096.867,221.963,427.789,177.507,17.695,152.278
C01357=1096.861,221.713,427.813,177.504,17.694,152.278
C01358=1096.855,221.465,427.838,177.500,17.693,152.279
C01359=1096.849,221.217,427.864,177.497,17.692,152.279
C01360=1096.844,220.967,427.889,177.493,17.691,152.279
C01361=1096.838,220.719,427.914,177.490,17.690,152.280
C01362=1096.832,220.470,427.938,177.487,17.689,152.280
C01363=1096.827,220.222,427.963,177.484,17.687,152.280
C01364=1096.821,219.973,427.989,177.481,17.686,152.281
C01365=1096.816,219.724,428.014,177.477,17.685,152.281
C01366=1096.810,219.476,428.039,177.474,17.684,152.282
C01367=1096.804,219.227,428.063,177.471,17.683,152.282
C01368=1096.798,218.978,428.088,177.467,17.682,152.282
C01369=1096.793,218.729,428.114,177.464,17.681,152.283
C01370=1096.787,218.481,428.139,177.460,17.680,152.283
C01371=1096.782,218.232,428.163,177.457,17.679,152.284
C01372=1096.776,217.984,428.188,177.455,17.677,152.284
C01373=1096.770,217.734,428.213,177.451,17.676,152.284
C01374=1096.764,217.486,428.238,177.448,17.675,152.285
C01375=1096.759,217.237,428.263,177.445,17.674,152.285
C01376=1096.754,216.988,428.287,177.441,17.673,152.285
C01377=1096.748,216.740,428.313,177.438,17.672,152.286
C01378=1096.742,216.491,428.337,177.435,17.671,152.286
C01379=1096.736,216.242,428.362,177.432,17.670,152.287
C01380=1096.731,215.994,428.386,177.429,17.669,152.287
C01381=1096.726,215.745,428.411,177.425,17.667,152.287
C01382=1096.720,215.496,428.437,177.422,17.666,152.288
C01383=1096.715,215.248,428.461,177.419,17.666,152.288
C01384=1096.709,214.998,428.486,177.415,17.664,152.288
C01385=1096.703,214.750,428.511,177.412,17.663,152.289
C01386=1096.697,214.501,428.535,177.409,17.663,152.289
C01387=1096.692,214.252,428.559,177.406,17.661,152.290
C01388=1096.687,214.004,428.584,177.403,17.660,152.290
C01389=1096.681,213.755,428.609,177.399,17.659,152.290
C01390=1096.675,213.507,428.633,177.396,17.658,152.291
C01391=1096.669,213.257,428.658,177.393,17.657,152.291
C01392=1096.664,213.009,428.683,177.390,17.655,152.292
C01393=1096.658,212.760,428.707,177.387,17.655,152.292
C01394=1096.653,212.511,428.732,177.384,17.654,152.292
C01395=1096.647,212.263,428.756,177.380,17.652,152.293
C01396=1096.641,212.014,428.781,177.377,17.652,152.293
C01397=1096.636,211.766,428.806,177.374,17.651,152.293
C01398=1096.630,211.516,428.830,177.370,17.649,152.294
C01399=1096.625,211.268,428.854,177.367,17.648,152.294
C01400=1096.619,211.019,428.879,177.364,17.647,152.295
C01401=1096.613,210.770,428.903,177.361,17.646,152.295
C01402=1096.608,210.521,428.928,177.358,17.645,152.295
C01403=1096.603,210.273,428.952,177.355,17.644,152.296
C01404=1096.597,210.023,428.976,177.351,17.643,152.296
C01405=1096.589,209.651,429.013,177.346,17.641,152.297
C01406=1096.580,209.279,429.049,177.341,17.640,152.297
C01407=1096.572,208.906,429.086,177.336,17.638,152.298
C01408=1096.563,208.534,429.122,177.332,17.637,152.299
C01409=1096.540,207.522,429.220,177.283,17.618,152.304
C01410=1096.535,207.273,429.244,177.279,17.617,152.304
C01411=1096.528,207.024,429.269,177.276,17.616,152.305
C01412=1096.523,206.775,429.292,177.272,17.617,152.306
C01413=1096.518,206.526,429.316,177.269,17.616,152.306
C01414=1096.512,206.278,429.340,177.265,17.616,152.307
C01415=1096.506,206.029,429.365,177.262,17.616,152.307
C01416=1096.501,205.779,429.388,177.259,17.616,152.308
C01417=1096.495,205.531,429.412,177.255,17.616,152.309
C01418=1096.490,205.283,429.436,177.252,17.615,152.309
C01419=1096.484,205.034,429.460,177.249,17.616,152.310
C01420=1096.478,204.784,429.484,177.245,17.615,152.310
C01421=1096.473,204.536,429.508,177.242,17.615,152.311
C01422=1096.467,204.287,429.532,177.239,17.615,152.312
C01423=1096.462,204.038,429.555,177.235,17.615,152.312
C01424=1096.457,203.790,429.579,177.232,17.614,152.313
C01425=1096.450,203.541,429.603,177.229,17.614,152.313
C01426=1096.445,203.292,429.627,177.225,17.614,152.314
C01427=1096.439,203.043,429.651,177.222,17.614,152.315
C01428=1096.434,202.794,429.674,177.219,17.614,152.315
C01429=1096.428,202.546,429.698,177.215,17.613,152.316
C01430=1096.423,202.297,429.722,177.212,17.614,152.317
C01431=1096.416,202.048,429.745,177.209,17.613,152.317
C01432=1096.411,201.799,429.770,177.205,17.613,152.318
C01433=1096.405,201.550,429.793,177.202,17.613,152.318
C01434=1096.399,201.302,429.816,177.199,17.613,152.319
C01435=1096.394,201.053,429.840,177.195,17.613,152.320
C01436=1096.387,200.804,429.864,177.192,17.612,152.320
C01437=1096.383,200.554,429.887,177.189,17.612,152.321
C01438=1096.376,200.306,429.911,177.185,17.612,152.321
C01439=1096.371,200.057,429.934,177.182,17.612,152.322
C01440=1096.365,199.809,429.958,177.178,17.612,152.323
C01441=1096.360,199.560,429.981,177.175,17.612,152.323
C01442=1096.354,199.311,430.005,177.172,17.611,152.324
C01443=1096.348,199.062,430.029,177.168,17.611,152.324
C01444=1096.342,198.813,430.052,177.165,17.611,152.325
C01445=1096.337,198.564,430.076,177.162,17.611,152.326
C01446=1096.331,198.316,430.100,177.158,17.611,152.326
C01447=1096.325,198.067,430.122,177.155,17.610,152.327
C01448=1096.320,197.818,430.146,177.152,17.610,152.327
C01449=1096.314,197.569,430.170,177.148,17.610,152.328
C01450=1096.309,197.321,430.193,177.145,17.610,152.329
C01451=1096.304,197.071,430.216,177.142,17.610,152.329
C01452=1096.297,196.823,430.240,177.138,17.609,152.330
C01453=1096.291,196.573,430.263,177.135,17.609,152.330
C01454=1096.286,196.324,430.287,177.132,17.609,152.331
C01455=1096.280,196.076,430.310,177.128,17.609,152.332
C01456=1096.274,195.827,430.333,177.125,17.609,152.332
C01457=1096.269,195.578,430.356,177.122,17.608,152.333
C01458=1096.263,195.330,430.381,177.118,17.608,152.333
C01459=1096.258,195.081,430.403,177.115,17.608,152.334
C01460=1096.252,194.832,430.426,177.112,17.608,152.335
C01461=1096.247,194.583,430.450,177.108,17.608,152.335
C01462=1096.241,194.334,430.473,177.105,17.607,152.336
C01463=1096.235,194.085,430.497,177.102,17.607,152.336
C01464=1096.229,193.837,430.519,177.099,17.607,152.337
C01465=1096.224,193.587,430.543,177.096,17.607,152.337
C01466=1096.219,193.338,430.566,177.093,17.607,152.338
C01467=1096.213,193.090,430.589,177.089,17.607,152.339
C01468=1096.207,192.841,430.613,177.086,17.606,152.339
C01469=1096.202,192.592,430.636,177.083,17.606,152.340
C01470=1096.196,192.318,430.661,177.079,17.605,152.340
C01471=1096.189,192.043,430.686,177.075,17.605,152.341
C01472=1096.184,191.768,430.712,177.072,17.605,152.342
C01473=1096.177,191.493,430.738,177.069,17.605,152.342
C01474=1096.171,191.245,430.761,177.065,17.605,152.343
C01475=1096.166,190.996,430.784,177.062,17.604,152.343
C01476=1096.160,190.747,430.807,177.059,17.604,152.344
C01477=1096.156,190.498,430.830,177.055,17.604,152.345
C01478=1096.150,190.249,430.853,177.052,17.604,152.345
C01479=1096.144,190.000,430.876,177.049,17.603,152.346
C01480=1096.138,189.752,430.899,177.046,17.603,152.346
C01481=1096.133,189.503,430.922,177.042,17.603,152.347
C01482=1096.128,189.253,430.945,177.039,17.602,152.347
C01483=1096.122,189.005,430.968,177.036,17.602,152.348
C01484=1096.116,188.756,430.991,177.033,17.602,152.348
C01485=1096.110,188.507,431.014,177.029,17.601,152.349
C01486=1096.105,188.259,431.036,177.026,17.601,152.350
C01487=1096.100,188.010,431.059,177.023,17.601,152.350
C01488=1096.094,187.761,431.082,177.020,17.600,152.351
C01489=1096.089,187.512,431.106,177.016,17.600,152.351
C01490=1096.083,187.263,431.129,177.013,17.600,152.352
C01491=1096.077,187.014,431.152,177.011,17.600,152.352
C01492=1096.072,186.765,431.175,177.007,17.600,152.353
C01493=1096.067,186.517,431.197,177.004,17.599,152.353
C01494=1096.061,186.267,431.220,177.001,17.599,152.354
C01495=1096.055,186.018,431.243,176.998,17.599,152.355
C01496=1096.050,185.769,431.265,176.994,17.598,152.355
C01497=1096.044,185.521,431.288,176.991,17.598,152.356
C01498=1096.040,185.272,431.312,176.988,17.598,152.356
C01499=1096.033,185.023,431.334,176.985,17.597,152.357
C01500=1096.028,184.774,431.356,176.981,17.598,152.357
C01501=1096.022,184.525,431.379,176.978,17.597,152.358
C01502=1096.016,184.276,431.402,176.975,17.597,152.359
C01503=1096.010,184.027,431.425,176.971,17.597,152.359
C01504=1096.004,183.778,431.447,176.968,17.596,152.360
C01505=1095.999,183.529,431.470,176.966,17.597,152.360
C01506=1095.993,183.280,431.493,176.962,17.596,152.361
C01507=1095.988,183.032,431.515,176.959,17.596,152.361
C01508=1095.982,182.782,431.537,176.956,17.596,152.362
C01509=1095.976,182.534,431.560,176.952,17.596,152.363
C01510=1095.970,182.285,431.583,176.949,17.595,152.363
C01511=1095.965,182.035,431.605,176.946,17.595,152.364
C01512=1095.959,181.787,431.628,176.943,17.595,152.364
C01513=1095.952,181.538,431.650,176.939,17.594,152.365
C01514=1095.948,181.289,431.672,176.936,17.594,152.365
C01515=1095.942,181.040,431.695,176.933,17.594,152.366
C01516=1095.936,180.791,431.718,176.930,17.594,152.366
C01517=1095.930,180.542,431.740,176.927,17.594,152.367
C01518=1095.924,180.293,431.763,176.924,17.593,152.368
C01519=1095.919,180.044,431.785,176.921,17.593,152.368
C01520=1095.914,179.796,431.807,176.917,17.593,152.369
C01521=1095.907,179.547,431.830,176.914,17.592,152.369
C01522=1095.902,179.297,431.852,176.911,17.592,152.370
C01523=1095.896,179.049,431.875,176.908,17.592,152.370
C01524=1095.890,178.799,431.896,176.904,17.592,152.371
C01525=1095.885,178.551,431.919,176.902,17.592,152.371
C01526=1095.879,178.302,431.941,176.899,17.591,152.372
C01527=1095.873,178.053,431.964,176.896,17.591,152.373
C01528=1095.867,177.804,431.986,176.892,17.591,152.373
C01529=1095.862,177.555,432.008,176.889,17.591,152.374
C01530=1095.856,177.306,432.030,176.886,17.590,152.374
C01531=1095.850,177.057,432.053,176.882,17.590,152.375
C01532=1095.845,176.808,432.075,176.879,17.590,152.375
C01533=1095.839,176.560,432.097,176.876,17.589,152.376
C01534=1095.833,176.284,432.122,176.873,17.589,152.376
C01535=1095.827,176.010,432.147,176.869,17.589,152.377
C01536=1095.821,175.734,432.171,176.866,17.588,152.378
C01537=1095.815,175.459,432.195,176.863,17.588,152.378
C01538=1095.808,175.211,432.218,176.860,17.588,152.379
C01539=1095.804,174.962,432.240,176.856,17.587,152.379
C01540=1095.797,174.713,432.261,176.853,17.587,152.380
C01541=1095.792,174.464,432.284,176.850,17.587,152.380
C01542=1095.787,174.215,432.306,176.847,17.586,152.381
C01543=1095.781,173.966,432.328,176.844,17.586,152.381
C01544=1095.775,173.717,432.351,176.841,17.586,152.382
C01545=1095.769,173.468,432.372,176.838,17.586,152.382
C01546=1095.764,173.219,432.394,176.835,17.585,152.383
C01547=1095.758,172.970,432.417,176.832,17.585,152.384
C01548=1095.753,172.721,432.438,176.828,17.585,152.384
C01549=1095.747,172.472,432.461,176.825,17.584,152.385
C01550=1095.742,172.223,432.482,176.822,17.584,152.385
C01551=1095.736,171.974,432.505,176.819,17.583,152.386
C01552=1095.730,171.725,432.526,176.816,17.584,152.386
C01553=1095.725,171.476,432.548,176.813,17.583,152.387
C01554=1095.720,171.227,432.571,176.810,17.582,152.387
C01555=1095.714,170.978,432.592,176.807,17.582,152.388
C01556=1095.708,170.729,432.615,176.804,17.582,152.388
C01557=1095.702,170.480,432.636,176.801,17.581,152.389
C01558=1095.697,170.231,432.658,176.797,17.581,152.389
C01559=1095.691,169.982,432.680,176.795,17.581,152.390
C01560=1095.686,169.733,432.702,176.792,17.580,152.390
C01561=1095.680,169.484,432.723,176.789,17.580,152.391
C01562=1095.675,169.235,432.745,176.785,17.580,152.391
C01563=1095.669,168.987,432.768,176.782,17.579,152.392
C01564=1095.663,168.737,432.790,176.779,17.579,152.392
C01565=1095.658,168.489,432.811,176.776,17.578,152.393
C01566=1095.652,168.239,432.833,176.774,17.578,152.393
C01567=1095.647,167.991,432.855,176.771,17.578,152.394
C01568=1095.641,167.741,432.877,176.767,17.577,152.394
C01569=1095.636,167.493,432.898,176.764,17.577,152.395
C01570=1095.630,167.243,432.920,176.761,17.576,152.395
C01571=1095.625,166.995,432.942,176.758,17.576,152.396
C01572=1095.619,166.745,432.964,176.755,17.575,152.396
C01573=1095.614,166.497,432.985,176.752,17.576,152.397
C01574=1095.609,166.247,433.007,176.749,17.575,152.397
C01575=1095.603,165.999,433.029,176.746,17.575,152.398
C01576=1095.597,165.749,433.050,176.743,17.574,152.398
C01577=1095.592,165.501,433.072,176.740,17.573,152.399
C01578=1095.586,165.252,433.093,176.737,17.573,152.399
C01579=1095.581,165.003,433.116,176.734,17.572,152.400
C01580=1095.575,164.754,433.137,176.731,17.573,152.400
C01581=1095.570,164.505,433.159,176.728,17.572,152.401
C01582=1095.565,164.255,433.180,176.725,17.572,152.401
C01583=1095.559,164.006,433.202,176.722,17.571,152.402
C01584=1095.554,163.757,433.223,176.719,17.571,152.402
C01585=1095.548,163.509,433.244,176.716,17.570,152.403
C01586=1095.543,163.259,433.267,176.713,17.570,152.403
C01587=1095.537,163.011,433.288,176.710,17.569,152.404
C01588=1095.532,162.761,433.310,176.707,17.569,152.404
C01589=1095.527,162.512,433.331,176.704,17.568,152.405
C01590=1095.521,162.264,433.352,176.701,17.567,152.405
C01591=1095.516,162.014,433.374,176.698,17.567,152.405
C01592=1095.510,161.766,433.395,176.696,17.567,152.406
C01593=1095.504,161.517,433.417,176.692,17.567,152.406
C01594=1095.499,161.267,433.438,176.689,17.566,152.407
C01595=1095.493,161.018,433.460,176.686,17.566,152.407
C01596=1095.488,160.769,433.481,176.683,17.565,152.408
C01597=1095.482,160.521,433.502,176.681,17.565,152.408
C01598=1095.475,160.245,433.526,176.677,17.564,152.409
C01599=1095.470,159.970,433.550,176.673,17.564,152.410
C01600=1095.463,159.695,433.573,176.670,17.564,152.410
C01601=1095.456,159.419,433.597,176.667,17.563,152.410
C01602=1095.452,159.170,433.618,176.664,17.563,152.411
C01603=1095.446,158.921,433.639,176.661,17.562,152.411
C01604=1095.440,158.672,433.661,176.658,17.562,152.412
C01605=1095.435,158.423,433.681,176.656,17.561,152.412
C01606=1095.429,158.174,433.703,176.652,17.561,152.413
C01607=1095.423,157.925,433.724,176.649,17.560,152.413
C01608=1095.417,157.675,433.745,176.646,17.560,152.414
C01609=1095.412,157.427,433.766,176.644,17.560,152.414
C01610=1095.406,157.178,433.788,176.641,17.560,152.415
C01611=1095.400,156.929,433.809,176.638,17.559,152.415
C01612=1095.396,156.680,433.830,176.635,17.558,152.416
C01613=1095.390,156.431,433.851,176.631,17.558,152.416
C01614=1095.384,156.181,433.873,176.629,17.558,152.417
C01615=1095.379,155.932,433.893,176.626,17.557,152.417
C01616=1095.373,155.684,433.914,176.623,17.556,152.418
C01617=1095.367,155.435,433.936,176.620,17.556,152.418
C01618=1095.362,155.186,433.957,176.617,17.555,152.419
C01619=1095.356,154.937,433.978,176.615,17.555,152.419
C01620=1095.350,154.687,433.999,176.611,17.555,152.420
C01621=1095.345,154.439,434.020,176.608,17.554,152.420
C01622=1095.339,154.189,434.041,176.605,17.554,152.421
C01623=1095.333,153.940,434.062,176.602,17.553,152.421
C01624=1095.328,153.691,434.083,176.600,17.553,152.421
C01625=1095.323,153.442,434.103,176.597,17.553,152.422
C01626=1095.317,153.193,434.125,176.594,17.552,152.422
C01627=1095.312,152.944,434.146,176.591,17.551,152.423
C01628=1095.306,152.695,434.167,176.587,17.551,152.423
C01629=1095.299,152.446,434.187,176.585,17.551,152.424
C01630=1095.294,152.197,434.208,176.582,17.550,152.424
C01631=1095.289,151.948,434.229,176.579,17.550,152.425
C01632=1095.283,151.698,434.250,176.576,17.549,152.425
C01633=1095.277,151.450,434.271,176.574,17.549,152.425
C01634=1095.272,151.201,434.292,176.571,17.548,152.426
C01635=1095.267,150.952,434.312,176.568,17.548,152.426
C01636=1095.260,150.702,434.334,176.565,17.547,152.427
C01637=1095.255,150.453,434.354,176.561,17.547,152.427
C01638=1095.250,150.204,434.375,176.559,17.546,152.428
C01639=1095.244,149.956,434.396,176.556,17.546,152.428
C01640=1095.238,149.706,434.417,176.553,17.545,152.429
C01641=1095.233,149.457,434.437,176.550,17.545,152.429
C01642=1095.227,149.208,434.458,176.548,17.544,152.430
C01643=1095.222,148.959,434.479,176.545,17.544,152.430
C01644=1095.216,148.709,434.500,176.542,17.543,152.430
C01645=1095.211,148.460,434.520,176.539,17.543,152.431
C01646=1095.204,148.212,434.541,176.536,17.542,152.431
C01647=1095.199,147.963,434.562,176.533,17.542,152.432
C01648=1095.193,147.713,434.583,176.530,17.541,152.432
C01649=1095.188,147.464,434.603,176.527,17.541,152.433
C01650=1095.182,147.215,434.623,176.524,17.540,152.433
C01651=1095.176,146.967,434.644,176.522,17.540,152.434
C01652=1095.171,146.718,434.665,176.519,17.539,152.434
C01653=1095.165,146.468,434.686,176.516,17.539,152.435
C01654=1095.159,146.219,434.706,176.513,17.538,152.435
C01655=1095.154,145.970,434.726,176.511,17.538,152.435
C01656=1095.149,145.721,434.747,176.508,17.537,152.436
C01657=1095.142,145.471,434.767,176.505,17.536,152.436
C01658=1095.137,145.223,434.789,176.501,17.536,152.437
C01659=1095.131,144.974,434.809,176.499,17.536,152.437
C01660=1095.126,144.725,434.830,176.496,17.535,152.438
C01661=1095.120,144.476,434.850,176.493,17.534,152.438
C01662=1095.114,144.200,434.872,176.490,17.534,152.439
C01663=1095.108,143.924,434.895,176.487,17.533,152.439
C01664=1095.102,143.648,434.918,176.484,17.532,152.439
C01665=1095.095,143.373,434.941,176.481,17.532,152.440
C01666=1095.089,143.124,434.961,176.478,17.531,152.440
C01667=1095.084,142.875,434.981,176.475,17.531,152.441
C01668=1095.079,142.626,435.002,176.473,17.531,152.441
C01669=1095.073,142.377,435.022,176.470,17.530,152.442
C01670=1095.068,142.128,435.042,176.467,17.529,152.442
C01671=1095.062,141.878,435.063,176.464,17.528,152.442
C01672=1095.056,141.630,435.083,176.461,17.528,152.443
C01673=1095.050,141.380,435.104,176.458,17.527,152.443
C01674=1095.045,141.131,435.124,176.455,17.527,152.444
C01675=1095.040,140.882,435.144,176.452,17.526,152.444
C01676=1095.034,140.633,435.164,176.450,17.526,152.444
C01677=1095.028,140.384,435.184,176.447,17.525,152.445
C01678=1095.023,140.135,435.205,176.444,17.525,152.445
C01679=1095.017,139.886,435.225,176.441,17.524,152.446
C01680=1095.011,139.636,435.245,176.439,17.524,152.446
C01681=1095.005,139.387,435.265,176.436,17.523,152.447
C01682=1095.000,139.138,435.286,176.433,17.522,152.447
C01683=1094.994,138.889,435.306,176.431,17.522,152.447
C01684=1094.989,138.640,435.326,176.428,17.521,152.448
C01685=1094.983,138.391,435.346,176.425,17.521,152.448
C01686=1094.978,138.142,435.366,176.422,17.520,152.449
C01687=1094.972,137.893,435.386,176.420,17.520,152.449
C01688=1094.966,137.644,435.407,176.417,17.519,152.449
C01689=1094.960,137.395,435.427,176.414,17.518,152.450
C01690=1094.956,137.145,435.447,176.411,17.517,152.450
C01691=1094.950,136.896,435.467,176.408,17.517,152.451
C01692=1094.944,136.647,435.487,176.405,17.516,152.451
C01693=1094.938,136.398,435.507,176.402,17.516,152.452
C01694=1094.933,136.149,435.527,176.400,17.516,152.452
C01695=1094.927,135.899,435.547,176.397,17.515,152.452
C01696=1094.921,135.650,435.567,176.394,17.514,152.453
C01697=1094.916,135.401,435.588,176.391,17.513,152.453
C01698=1094.910,135.152,435.607,176.389,17.513,152.454
C01699=1094.905,134.903,435.628,176.386,17.512,152.454
C01700=1094.899,134.654,435.648,176.383,17.511,152.454
C01701=1094.893,134.404,435.667,176.381,17.511,152.455
C01702=1094.888,134.155,435.687,176.378,17.510,152.455
C01703=1094.882,133.907,435.707,176.375,17.509,152.455
C01704=1094.877,133.657,435.727,176.372,17.509,152.456
C01705=1094.871,133.408,435.747,176.370,17.509,152.456
C01706=1094.865,133.159,435.767,176.367,17.508,152.457
C01707=1094.860,132.909,435.787,176.364,17.507,152.457
C01708=1094.854,132.661,435.806,176.362,17.506,152.457
C01709=1094.849,132.412,435.826,176.359,17.506,152.458
C01710=1094.843,132.163,435.846,176.356,17.505,152.458
C01711=1094.837,131.914,435.866,176.353,17.504,152.459
C01712=1094.832,131.665,435.885,176.351,17.504,152.459
C01713=1094.826,131.416,435.905,176.348,17.503,152.459
C01714=1094.821,131.166,435.925,176.345,17.503,152.460
C01715=1094.814,130.916,435.946,176.343,17.502,152.460
C01716=1094.809,130.668,435.964,176.340,17.502,152.461
C01717=1094.803,130.419,435.984,176.337,17.500,152.461
C01718=1094.797,130.169,436.004,176.334,17.500,152.461
C01719=1094.791,129.921,436.024,176.332,17.499,152.462
C01720=1094.786,129.672,436.044,176.329,17.499,152.462
C01721=1094.780,129.422,436.063,176.326,17.498,152.463
C01722=1094.775,129.173,436.083,176.324,17.498,152.463
C01723=1094.769,128.924,436.103,176.321,17.497,152.463
C01724=1094.763,128.674,436.122,176.318,17.496,152.464
C01725=1094.757,128.426,436.142,176.316,17.496,152.464
C01726=1094.751,128.149,436.164,176.313,17.495,152.464
C01727=1094.745,127.874,436.186,176.310,17.494,152.465
C01728=1094.738,127.598,436.207,176.307,17.493,152.465
C01729=1094.732,127.323,436.229,176.304,17.493,152.466
C01730=1094.727,127.073,436.249,176.301,17.492,152.466
C01731=1094.721,126.824,436.268,176.298,17.491,152.467
C01732=1094.715,126.575,436.288,176.296,17.491,152.467
C01733=1094.709,126.325,436.307,176.293,17.490,152.467
C01734=1094.704,126.077,436.327,176.290,17.489,152.468
C01735=1094.698,125.828,436.346,176.288,17.489,152.468
C01736=1094.693,125.578,436.365,176.285,17.488,152.468
C01737=1094.687,125.330,436.385,176.282,17.487,152.469
C01738=1094.681,125.080,436.404,176.280,17.487,152.469
C01739=1094.676,124.830,436.424,176.277,17.486,152.469
C01740=1094.670,124.582,436.444,176.275,17.485,152.470
C01741=1094.664,124.332,436.463,176.272,17.485,152.470
C01742=1094.659,124.083,436.482,176.269,17.484,152.471
C01743=1094.653,123.834,436.501,176.267,17.483,152.471
C01744=1094.647,123.585,436.521,176.264,17.483,152.471
C01745=1094.642,123.336,436.541,176.261,17.482,152.472
C01746=1094.636,123.086,436.560,176.259,17.481,152.472
C01747=1094.630,122.837,436.579,176.256,17.480,152.472
C01748=1094.625,122.589,436.599,176.254,17.480,152.473
C01749=1094.619,122.339,436.618,176.251,17.479,152.473
C01750=1094.614,122.090,436.637,176.248,17.478,152.473
C01751=1094.608,121.841,436.656,176.246,17.477,152.474
C01752=1094.602,121.591,436.676,176.243,17.476,152.474
C01753=1094.597,121.342,436.695,176.240,17.476,152.474
C01754=1094.591,121.094,436.714,176.238,17.475,152.475
C01755=1094.585,120.844,436.734,176.235,17.474,152.475
C01756=1094.580,120.595,436.753,176.232,17.473,152.475
C01757=1094.574,120.345,436.772,176.230,17.473,152.476
C01758=1094.569,120.097,436.791,176.228,17.472,152.476
C01759=1094.563,119.847,436.810,176.225,17.471,152.476
C01760=1094.558,119.598,436.830,176.223,17.470,152.477
C01761=1094.552,119.348,436.849,176.220,17.470,152.477
C01762=1094.547,119.099,436.868,176.217,17.468,152.477
C01763=1094.541,118.851,436.888,176.215,17.468,152.478
C01764=1094.535,118.601,436.907,176.212,17.467,152.478
C01765=1094.530,118.352,436.926,176.209,17.466,152.478
C01766=1094.524,118.103,436.945,176.207,17.466,152.479
C01767=1094.519,117.854,436.964,176.204,17.465,152.479
C01768=1094.513,117.604,436.984,176.201,17.464,152.479
C01769=1094.508,117.355,437.002,176.199,17.463,152.480
C01770=1094.502,117.106,437.022,176.197,17.462,152.480
C01771=1094.497,116.857,437.041,176.194,17.462,152.480
C01772=1094.492,116.608,437.060,176.192,17.461,152.481
C01773=1094.486,116.358,437.079,176.189,17.460,152.481
C01774=1094.480,116.109,437.098,176.187,17.460,152.481
C01775=1094.474,115.860,437.117,176.184,17.458,152.482
C01776=1094.469,115.611,437.136,176.181,17.458,152.482
C01777=1094.464,115.361,437.155,176.179,17.457,152.482
C01778=1094.458,115.112,437.174,176.176,17.456,152.483
C01779=1094.452,114.863,437.192,176.173,17.455,152.483
C01780=1094.447,114.614,437.212,176.172,17.454,152.483
C01781=1094.442,114.365,437.231,176.169,17.454,152.484
C01782=1094.436,114.115,437.250,176.166,17.452,152.484
C01783=1094.430,113.866,437.269,176.164,17.452,152.484
C01784=1094.424,113.617,437.288,176.161,17.451,152.485
C01785=1094.419,113.368,437.307,176.158,17.450,152.485
C01786=1094.413,113.118,437.325,176.156,17.450,152.485
C01787=1094.408,112.869,437.344,176.153,17.448,152.486
C01788=1094.402,112.620,437.363,176.150,17.448,152.486
C01789=1094.396,112.371,437.382,176.148,17.447,152.486
C01790=1094.390,112.095,437.403,176.145,17.446,152.487
C01791=1094.384,111.820,437.424,176.143,17.445,152.487
C01792=1094.378,111.543,437.444,176.140,17.444,152.487
C01793=1094.371,111.268,437.465,176.137,17.443,152.488
C01794=1094.366,111.019,437.484,176.135,17.443,152.488
C01795=1094.360,110.769,437.503,176.132,17.442,152.488
C01796=1094.354,110.520,437.521,176.129,17.441,152.489
C01797=1094.349,110.271,437.540,176.127,17.440,152.489
C01798=1094.343,110.021,437.559,176.124,17.439,152.489
C01799=1094.337,109.773,437.577,176.122,17.438,152.490
C01800=1094.332,109.523,437.596,176.120,17.438,152.490
C01801=1094.325,109.274,437.615,176.117,17.437,152.490
C01802=1094.320,109.025,437.633,176.115,17.436,152.491
C01803=1094.315,108.775,437.652,176.112,17.435,152.491
C01804=1094.309,108.526,437.671,176.109,17.434,152.491
C01805=1094.303,108.277,437.690,176.107,17.434,152.491
